LIN {X 0,Y 198.688,Z 628.366,A -85,B 0,C 180,E1 -21497.744,E2 -21497.744} C_VEL
LIN {X 0,Y 197.64,Z 631.779,A -85,B 0,C 180,E1 -21501.82,E2 -21501.82} C_VEL
LIN {X 0,Y 197.241,Z 633.877,A -85,B 0,C 180,E1 -21506.105,E2 -21506.105} C_VEL
LIN {X 0,Y 197.208,Z 634.499,A -85,B 0,C 180,E1 -21509.997,E2 -21509.997} C_VEL
LIN {X 0,Y 197.249,Z 633.864,A -85,B 0,C 180,E1 -21514.084,E2 -21514.084} C_VEL
LIN {X 0,Y 197.637,Z 631.888,A -85,B 0,C 180,E1 -21518.175,E2 -21518.175} C_VEL
LIN {X 0,Y 198.663,Z 628.524,A -85,B 0,C 180,E1 -21522.252,E2 -21522.252} C_VEL
LIN {X 0,Y 200.478,Z 623.671,A -85,B 0,C 180,E1 -21526.284,E2 -21526.284} C_VEL
LIN {X 0,Y 202.386,Z 618.993,A -85,B 0,C 180,E1 -21529.259,E2 -21529.259} C_VEL
LIN {X 0,Y 205.088,Z 612.195,A -85,B 0,C 180,E1 -21532.673,E2 -21532.673} C_VEL
LIN {X 0,Y 208.544,Z 603.751,A -85,B 0,C 180,E1 -21535.98,E2 -21535.98} C_VEL
LIN {X 0,Y 212.007,Z 594.94,A -85,B 0,C 180,E1 -21538.726,E2 -21538.726} C_VEL
LIN {X 0,Y 215.999,Z 584.265,A -85,B 0,C 180,E1 -21541.369,E2 -21541.369} C_VEL
LIN {X 0,Y 219.78,Z 572.903,A -85,B 0,C 180,E1 -21543.607,E2 -21543.607} C_VEL
LIN {X 0,Y 223.02,Z 561.657,A -85,B 0,C 180,E1 -21545.381,E2 -21545.381} C_VEL
LIN {X 0,Y 226.311,Z 548.608,A -85,B 0,C 180,E1 -21546.987,E2 -21546.987} C_VEL
LIN {X 0,Y 228.918,Z 536.079,A -85,B 0,C 180,E1 -21548.157,E2 -21548.157} C_VEL
LIN {X 0,Y 230.973,Z 522.952,A -85,B 0,C 180,E1 -21549.078,E2 -21549.078} C_VEL
LIN {X 0,Y 232.584,Z 508.808,A -85,B 0,C 180,E1 -21549.736,E2 -21549.736} C_VEL
LIN {X 0,Y 236.354,Z 442.048,A -85,B 0,C 180,E1 -21551.632,E2 -21551.632} C_VEL
LIN {X 0,Y 236.321,Z 438.308,A -85,B 0,C 180,E1 -21551.788,E2 -21551.788} C_VEL
LIN {X 0,Y 230.698,Z 425.066,A -85,B 0,C 180,E1 -21553.603,E2 -21553.603} C_VEL
LIN {X 0,Y 225.025,Z 413.286,A -85,B 0,C 180,E1 -21555.516,E2 -21555.516} C_VEL
LIN {X 0,Y 218.681,Z 401.679,A -85,B 0,C 180,E1 -21557.787,E2 -21557.787} C_VEL
LIN {X 0,Y 213.141,Z 392.925,A -85,B 0,C 180,E1 -21559.9,E2 -21559.9} C_VEL
LIN {X 0,Y 210.045,Z 388.672,A -85,B 0,C 180,E1 -21561.139,E2 -21561.139} C_VEL
LIN {X 0,Y 207.427,Z 384.974,A -85,B 0,C 180,E1 -21562.249,E2 -21562.249} C_VEL
LIN {X 0,Y 204.423,Z 381.506,A -85,B 0,C 180,E1 -21563.55,E2 -21563.55} C_VEL
LIN {X 0,Y 203.246,Z 379.556,A -85,B 0,C 180,E1 -21564.116,E2 -21564.116} C_VEL
LIN {X 0,Y 200.84,Z 377.317,A -85,B 0,C 180,E1 -21565.212,E2 -21565.212} C_VEL
LIN {X 0,Y 199.725,Z 374.788,A -85,B 0,C 180,E1 -21566.001,E2 -21566.001} C_VEL
LIN {X 0,Y 199.638,Z 374.276,A -85,B 0,C 180,E1 -21566.514,E2 -21566.514} C_VEL
LIN {X 0,Y 199.656,Z 374.162,A -85,B 0,C 180,E1 -21570.475,E2 -21570.475} C_VEL
LIN {X 0,Y 199.665,Z 374.22,A -85,B 0,C 180,E1 -21575.014,E2 -21575.014} C_VEL
LIN {X 0,Y 199.691,Z 374.213,A -85,B 0,C 180,E1 -21579.394,E2 -21579.394} C_VEL
LIN {X 0,Y 199.795,Z 374.197,A -85,B 0,C 180,E1 -21583.656,E2 -21583.656} C_VEL
LIN {X 0,Y 199.905,Z 374.205,A -85,B 0,C 180,E1 -21587.822,E2 -21587.822} C_VEL
LIN {X 0,Y 200.11,Z 374.161,A -85,B 0,C 180,E1 -21591.924,E2 -21591.924} C_VEL
LIN {X 0,Y 200.314,Z 374.135,A -85,B 0,C 180,E1 -21597.989,E2 -21597.989} C_VEL
LIN {X 0,Y 200.478,Z 374.139,A -85,B 0,C 180,E1 -21600,E2 -21600} C_VEL
LIN {X 0,Y 200.023,Z 374.168,A -85,B 0,C 180,E1 -21604.029,E2 -21604.029} C_VEL
LIN {X 0,Y 200.11,Z 374.161,A -85,B 0,C 180,E1 -21608.076,E2 -21608.076} C_VEL
LIN {X 0,Y 199.904,Z 374.203,A -85,B 0,C 180,E1 -21612.177,E2 -21612.177} C_VEL
LIN {X 0,Y 199.795,Z 374.195,A -85,B 0,C 180,E1 -21616.344,E2 -21616.344} C_VEL
LIN {X 0,Y 199.686,Z 374.214,A -85,B 0,C 180,E1 -21620.001,E2 -21620.001} C_VEL
LIN {X 0,Y 199.025,Z 374.304,A -85,B 0,C 180,E1 -21621.684,E2 -21621.684} C_VEL
LIN {X 0,Y 196.217,Z 374.664,A -85,B 0,C 180,E1 -21624.437,E2 -21624.437} C_VEL
LIN {X 0,Y 192.97,Z 374.996,A -85,B 0,C 180,E1 -21627.849,E2 -21627.849} C_VEL
LIN {X 0,Y 192.61,Z 375.041,A -85,B 0,C 180,E1 -21629.032,E2 -21629.032} C_VEL
LIN {X 0,Y 192.647,Z 375.427,A -85,B 0,C 180,E1 -21630.713,E2 -21630.713} C_VEL
LIN {X 0,Y 193.159,Z 377.057,A -85,B 0,C 180,E1 -21631.383,E2 -21631.383} C_VEL
LIN {X 0,Y 195.117,Z 379.67,A -85,B 0,C 180,E1 -21632.495,E2 -21632.495} C_VEL
LIN {X 0,Y 196.745,Z 380.901,A -85,B 0,C 180,E1 -21633.313,E2 -21633.313} C_VEL
LIN {X 0,Y 198.74,Z 384.113,A -85,B 0,C 180,E1 -21634.381,E2 -21634.381} C_VEL
LIN {X 0,Y 200.861,Z 386.283,A -85,B 0,C 180,E1 -21635.388,E2 -21635.388} C_VEL
LIN {X 0,Y 203.398,Z 389.783,A -85,B 0,C 180,E1 -21636.586,E2 -21636.586} C_VEL
LIN {X 0,Y 204.689,Z 391.4,A -85,B 0,C 180,E1 -21637.163,E2 -21637.163} C_VEL
LIN {X 0,Y 208.318,Z 396.435,A -85,B 0,C 180,E1 -21638.734,E2 -21638.734} C_VEL
LIN {X 0,Y 211.143,Z 400.453,A -85,B 0,C 180,E1 -21639.89,E2 -21639.89} C_VEL
LIN {X 0,Y 217.685,Z 411.697,A -85,B 0,C 180,E1 -21642.451,E2 -21642.451} C_VEL
LIN {X 0,Y 224.176,Z 424.655,A -85,B 0,C 180,E1 -21644.816,E2 -21644.816} C_VEL
LIN {X 0,Y 230.432,Z 439.17,A -85,B 0,C 180,E1 -21646.971,E2 -21646.971} C_VEL
LIN {X 0,Y 231.097,Z 440.853,A -85,B 0,C 180,E1 -21647.195,E2 -21647.195} C_VEL
LIN {X 0,Y 228.019,Z 496.452,A -85,B 0,C 180,E1 -21648.796,E2 -21648.796} C_VEL
LIN {X 0,Y 226.809,Z 513.234,A -85,B 0,C 180,E1 -21649.366,E2 -21649.366} C_VEL
LIN {X 0,Y 224.799,Z 527.804,A -85,B 0,C 180,E1 -21650.144,E2 -21650.144} C_VEL
LIN {X 0,Y 222.26,Z 541.368,A -85,B 0,C 180,E1 -21651.212,E2 -21651.212} C_VEL
LIN {X 0,Y 219.441,Z 553.628,A -85,B 0,C 180,E1 -21652.522,E2 -21652.522} C_VEL
LIN {X 0,Y 216.105,Z 565.698,A -85,B 0,C 180,E1 -21654.173,E2 -21654.173} C_VEL
LIN {X 0,Y 212.305,Z 577.878,A -85,B 0,C 180,E1 -21656.328,E2 -21656.328} C_VEL
LIN {X 0,Y 208.578,Z 587.941,A -85,B 0,C 180,E1 -21658.519,E2 -21658.519} C_VEL
LIN {X 0,Y 204.604,Z 597.944,A -85,B 0,C 180,E1 -21661.26,E2 -21661.26} C_VEL
LIN {X 0,Y 201.059,Z 606.25,A -85,B 0,C 180,E1 -21664.094,E2 -21664.094} C_VEL
LIN {X 0,Y 198.096,Z 613.182,A -85,B 0,C 180,E1 -21667.033,E2 -21667.033} C_VEL
LIN {X 0,Y 195.695,Z 618.917,A -85,B 0,C 180,E1 -21670.055,E2 -21670.055} C_VEL
LIN {X 0,Y 193.677,Z 623.61,A -85,B 0,C 180,E1 -21673.127,E2 -21673.127} C_VEL
LIN {X 0,Y 191.707,Z 628.478,A -85,B 0,C 180,E1 -21677.296,E2 -21677.296} C_VEL
LIN {X 0,Y 190.577,Z 631.857,A -85,B 0,C 180,E1 -21681.52,E2 -21681.52} C_VEL
LIN {X 0,Y 190.163,Z 633.848,A -85,B 0,C 180,E1 -21685.764,E2 -21685.764} C_VEL
LIN {X 0,Y 190.118,Z 634.5,A -85,B 0,C 180,E1 -21690.003,E2 -21690.003} C_VEL
LIN {X 0,Y 190.164,Z 633.824,A -85,B 0,C 180,E1 -21694.242,E2 -21694.242} C_VEL
LIN {X 0,Y 190.734,Z 631.811,A -85,B 0,C 180,E1 -21698.478,E2 -21698.478} C_VEL
LIN {X 0,Y 191.198,Z 630.901,A -85,B 0,C 180,E1 -21700.058,E2 -21700.058} C_VEL
LIN {X 0,Y 192.096,Z 632.211,A -85,B 0,C 180,E1 -21702.683,E2 -21702.683} C_VEL
LIN {X 0,Y 194.442,Z 633.199,A -85,B 0,C 180,E1 -21706.81,E2 -21706.81} C_VEL
LIN {X 0,Y 197.98,Z 632.816,A -85,B 0,C 180,E1 -21710.795,E2 -21710.795} C_VEL
LIN {X 0,Y 202.531,Z 631.063,A -85,B 0,C 180,E1 -21714.611,E2 -21714.611} C_VEL
LIN {X 0,Y 208.298,Z 627.892,A -85,B 0,C 180,E1 -21718.19,E2 -21718.19} C_VEL
LIN {X 0,Y 215.076,Z 623.289,A -85,B 0,C 180,E1 -21721.525,E2 -21721.525} C_VEL
LIN {X 0,Y 222.681,Z 617.112,A -85,B 0,C 180,E1 -21724.62,E2 -21724.62} C_VEL
LIN {X 0,Y 230.147,Z 610.231,A -85,B 0,C 180,E1 -21727.095,E2 -21727.095} C_VEL
LIN {X 0,Y 238.456,Z 601.514,A -85,B 0,C 180,E1 -21729.46,E2 -21729.46} C_VEL
LIN {X 0,Y 246.697,Z 591.63,A -85,B 0,C 180,E1 -21731.482,E2 -21731.482} C_VEL
LIN {X 0,Y 253.123,Z 582.904,A -85,B 0,C 180,E1 -21732.865,E2 -21732.865} C_VEL
LIN {X 0,Y 260.597,Z 571.402,A -85,B 0,C 180,E1 -21734.255,E2 -21734.255} C_VEL
LIN {X 0,Y 267.543,Z 558.852,A -85,B 0,C 180,E1 -21735.409,E2 -21735.409} C_VEL
LIN {X 0,Y 268.161,Z 557.592,A -85,B 0,C 180,E1 -21735.507,E2 -21735.507} C_VEL
LIN {X 0,Y 267.786,Z 558.493,A -85,B 0,C 180,E1 -21735.934,E2 -21735.934} C_VEL
LIN {X 0,Y 261.439,Z 570.62,A -85,B 0,C 180,E1 -21736.936,E2 -21736.936} C_VEL
LIN {X 0,Y 254.824,Z 581.361,A -85,B 0,C 180,E1 -21738.132,E2 -21738.132} C_VEL
LIN {X 0,Y 248.472,Z 590.482,A -85,B 0,C 180,E1 -21739.417,E2 -21739.417} C_VEL
LIN {X 0,Y 240.901,Z 599.981,A -85,B 0,C 180,E1 -21741.154,E2 -21741.154} C_VEL
LIN {X 0,Y 232.636,Z 609.079,A -85,B 0,C 180,E1 -21743.37,E2 -21743.37} C_VEL
LIN {X 0,Y 227.128,Z 614.466,A -85,B 0,C 180,E1 -21745.079,E2 -21745.079} C_VEL
LIN {X 0,Y 220.859,Z 619.969,A -85,B 0,C 180,E1 -21747.251,E2 -21747.251} C_VEL
LIN {X 0,Y 213.286,Z 625.729,A -85,B 0,C 180,E1 -21750.379,E2 -21750.379} C_VEL
LIN {X 0,Y 206.666,Z 629.831,A -85,B 0,C 180,E1 -21753.763,E2 -21753.763} C_VEL
LIN {X 0,Y 203.739,Z 631.338,A -85,B 0,C 180,E1 -21755.547,E2 -21755.547} C_VEL
LIN {X 0,Y 198.992,Z 633.231,A -85,B 0,C 180,E1 -21759.318,E2 -21759.318} C_VEL
LIN {X 0,Y 195.229,Z 633.698,A -85,B 0,C 180,E1 -21763.263,E2 -21763.263} C_VEL
LIN {X 0,Y 192.575,Z 632.768,A -85,B 0,C 180,E1 -21767.352,E2 -21767.352} C_VEL
LIN {X 0,Y 191.078,Z 630.391,A -85,B 0,C 180,E1 -21771.54,E2 -21771.54} C_VEL
LIN {X 0,Y 190.649,Z 626.452,A -85,B 0,C 180,E1 -21775.772,E2 -21775.772} C_VEL
LIN {X 0,Y 190.738,Z 622.348,A -85,B 0,C 180,E1 -21778.945,E2 -21778.945} C_VEL
LIN {X 0,Y 190.954,Z 617.045,A -85,B 0,C 180,E1 -21782.109,E2 -21782.109} C_VEL
LIN {X 0,Y 191.191,Z 610.328,A -85,B 0,C 180,E1 -21785.273,E2 -21785.273} C_VEL
LIN {X 0,Y 191.602,Z 601.884,A -85,B 0,C 180,E1 -21788.437,E2 -21788.437} C_VEL
LIN {X 0,Y 192.123,Z 593.245,A -85,B 0,C 180,E1 -21791.073,E2 -21791.073} C_VEL
LIN {X 0,Y 192.927,Z 582.773,A -85,B 0,C 180,E1 -21793.697,E2 -21793.697} C_VEL
LIN {X 0,Y 193.92,Z 571.144,A -85,B 0,C 180,E1 -21796.042,E2 -21796.042} C_VEL
LIN {X 0,Y 194.965,Z 558.197,A -85,B 0,C 180,E1 -21798.114,E2 -21798.114} C_VEL
LIN {X 0,Y 195.925,Z 544.563,A -85,B 0,C 180,E1 -21799.788,E2 -21799.788} C_VEL
LIN {X 0,Y 196.902,Z 529.324,A -85,B 0,C 180,E1 -21801.134,E2 -21801.134} C_VEL
LIN {X 0,Y 200.175,Z 458.461,A -85,B 0,C 180,E1 -21805.683,E2 -21805.683} C_VEL
LIN {X 0,Y 197.937,Z 429.916,A -85,B 0,C 180,E1 -21807.561,E2 -21807.561} C_VEL
LIN {X 0,Y 197.856,Z 419.514,A -85,B 0,C 180,E1 -21808.293,E2 -21808.293} C_VEL
LIN {X 0,Y 199.54,Z 406.784,A -85,B 0,C 180,E1 -21811.595,E2 -21811.595} C_VEL
LIN {X 0,Y 197.743,Z 398.022,A -85,B 0,C 180,E1 -21814.148,E2 -21814.148} C_VEL
LIN {X 0,Y 197.668,Z 397.343,A -85,B 0,C 180,E1 -21814.672,E2 -21814.672} C_VEL
LIN {X 0,Y 198.255,Z 397.732,A -85,B 0,C 180,E1 -21815.174,E2 -21815.174} C_VEL
LIN {X 0,Y 199.201,Z 398.055,A -85,B 0,C 180,E1 -21815.601,E2 -21815.601} C_VEL
LIN {X 0,Y 201.049,Z 397.617,A -85,B 0,C 180,E1 -21816.305,E2 -21816.305} C_VEL
LIN {X 0,Y 202.414,Z 396.833,A -85,B 0,C 180,E1 -21816.783,E2 -21816.783} C_VEL
LIN {X 0,Y 203.399,Z 397.137,A -85,B 0,C 180,E1 -21817.17,E2 -21817.17} C_VEL
LIN {X 0,Y 206.725,Z 396.78,A -85,B 0,C 180,E1 -21818.351,E2 -21818.351} C_VEL
LIN {X 0,Y 208.167,Z 396.459,A -85,B 0,C 180,E1 -21818.833,E2 -21818.833} C_VEL
LIN {X 0,Y 211.293,Z 400.891,A -85,B 0,C 180,E1 -21820.105,E2 -21820.105} C_VEL
LIN {X 0,Y 217.272,Z 411.228,A -85,B 0,C 180,E1 -21822.442,E2 -21822.442} C_VEL
LIN {X 0,Y 222.993,Z 422.302,A -85,B 0,C 180,E1 -21824.527,E2 -21824.527} C_VEL
LIN {X 0,Y 229.105,Z 435.988,A -85,B 0,C 180,E1 -21826.643,E2 -21826.643} C_VEL
LIN {X 0,Y 230.998,Z 440.808,A -85,B 0,C 180,E1 -21827.285,E2 -21827.285} C_VEL
LIN {X 0,Y 227.011,Z 509.642,A -85,B 0,C 180,E1 -21829.293,E2 -21829.293} C_VEL
LIN {X 0,Y 225.229,Z 524.29,A -85,B 0,C 180,E1 -21830.011,E2 -21830.011} C_VEL
LIN {X 0,Y 222.752,Z 538.201,A -85,B 0,C 180,E1 -21831.018,E2 -21831.018} C_VEL
LIN {X 0,Y 219.914,Z 551.142,A -85,B 0,C 180,E1 -21832.321,E2 -21832.321} C_VEL
LIN {X 0,Y 216.535,Z 563.696,A -85,B 0,C 180,E1 -21833.963,E2 -21833.963} C_VEL
LIN {X 0,Y 212.694,Z 576.322,A -85,B 0,C 180,E1 -21836.108,E2 -21836.108} C_VEL
LIN {X 0,Y 208.627,Z 587.578,A -85,B 0,C 180,E1 -21838.521,E2 -21838.521} C_VEL
LIN {X 0,Y 204.647,Z 597.642,A -85,B 0,C 180,E1 -21841.261,E2 -21841.261} C_VEL
LIN {X 0,Y 201.12,Z 605.999,A -85,B 0,C 180,E1 -21844.097,E2 -21844.097} C_VEL
LIN {X 0,Y 198.086,Z 612.973,A -85,B 0,C 180,E1 -21847.026,E2 -21847.026} C_VEL
LIN {X 0,Y 195.695,Z 618.734,A -85,B 0,C 180,E1 -21850.049,E2 -21850.049} C_VEL
LIN {X 0,Y 193.689,Z 623.467,A -85,B 0,C 180,E1 -21853.123,E2 -21853.123} C_VEL
LIN {X 0,Y 191.72,Z 628.367,A -85,B 0,C 180,E1 -21857.292,E2 -21857.292} C_VEL
LIN {X 0,Y 190.581,Z 631.779,A -85,B 0,C 180,E1 -21861.515,E2 -21861.515} C_VEL
LIN {X 0,Y 190.165,Z 633.807,A -85,B 0,C 180,E1 -21865.758,E2 -21865.758} C_VEL
LIN {X 0,Y 190.119,Z 634.499,A -85,B 0,C 180,E1 -21869.997,E2 -21869.997} C_VEL
LIN {X 0,Y 190.164,Z 633.863,A -85,B 0,C 180,E1 -21874.236,E2 -21874.236} C_VEL
LIN {X 0,Y 190.578,Z 631.888,A -85,B 0,C 180,E1 -21878.48,E2 -21878.48} C_VEL
LIN {X 0,Y 191.697,Z 628.523,A -85,B 0,C 180,E1 -21882.705,E2 -21882.705} C_VEL
LIN {X 0,Y 193.643,Z 623.669,A -85,B 0,C 180,E1 -21886.876,E2 -21886.876} C_VEL
LIN {X 0,Y 196.435,Z 617.183,A -85,B 0,C 180,E1 -21890.961,E2 -21890.961} C_VEL
LIN {X 0,Y 199.479,Z 609.962,A -85,B 0,C 180,E1 -21894.452,E2 -21894.452} C_VEL
LIN {X 0,Y 203.313,Z 601.028,A -85,B 0,C 180,E1 -21897.815,E2 -21897.815} C_VEL
LIN {X 0,Y 207.088,Z 591.645,A -85,B 0,C 180,E1 -21900.598,E2 -21900.598} C_VEL
LIN {X 0,Y 211.056,Z 581.254,A -85,B 0,C 180,E1 -21903.04,E2 -21903.04} C_VEL
LIN {X 0,Y 214.822,Z 569.884,A -85,B 0,C 180,E1 -21905.189,E2 -21905.189} C_VEL
LIN {X 0,Y 218.525,Z 557.084,A -85,B 0,C 180,E1 -21907.083,E2 -21907.083} C_VEL
LIN {X 0,Y 221.531,Z 544.705,A -85,B 0,C 180,E1 -21908.503,E2 -21908.503} C_VEL
LIN {X 0,Y 223.986,Z 532.273,A -85,B 0,C 180,E1 -21909.591,E2 -21909.591} C_VEL
LIN {X 0,Y 226.11,Z 518.478,A -85,B 0,C 180,E1 -21910.451,E2 -21910.451} C_VEL
LIN {X 0,Y 227.577,Z 504,A -85,B 0,C 180,E1 -21911.025,E2 -21911.025} C_VEL
LIN {X 0,Y 231.081,Z 440.795,A -85,B 0,C 180,E1 -21912.856,E2 -21912.856} C_VEL
LIN {X 0,Y 225.276,Z 427.11,A -85,B 0,C 180,E1 -21914.84,E2 -21914.84} C_VEL
LIN {X 0,Y 219.25,Z 414.668,A -85,B 0,C 180,E1 -21917.009,E2 -21917.009} C_VEL
LIN {X 0,Y 212.764,Z 403.025,A -85,B 0,C 180,E1 -21919.504,E2 -21919.504} C_VEL
LIN {X 0,Y 209.554,Z 398.139,A -85,B 0,C 180,E1 -21920.801,E2 -21920.801} C_VEL
LIN {X 0,Y 206.285,Z 393.654,A -85,B 0,C 180,E1 -21922.175,E2 -21922.175} C_VEL
LIN {X 0,Y 203.588,Z 389.967,A -85,B 0,C 180,E1 -21923.376,E2 -21923.376} C_VEL
LIN {X 0,Y 200.923,Z 386.44,A -85,B 0,C 180,E1 -21924.623,E2 -21924.623} C_VEL
LIN {X 0,Y 200.029,Z 385.368,A -85,B 0,C 180,E1 -21925.05,E2 -21925.05} C_VEL
LIN {X 0,Y 197.51,Z 382.418,A -85,B 0,C 180,E1 -21926.298,E2 -21926.298} C_VEL
LIN {X 0,Y 196.601,Z 380.655,A -85,B 0,C 180,E1 -21926.812,E2 -21926.812} C_VEL
LIN {X 0,Y 194.197,Z 378.704,A -85,B 0,C 180,E1 -21928.045,E2 -21928.045} C_VEL
LIN {X 0,Y 192.706,Z 375.703,A -85,B 0,C 180,E1 -21929.145,E2 -21929.145} C_VEL
LIN {X 0,Y 192.613,Z 375.156,A -85,B 0,C 180,E1 -21929.791,E2 -21929.791} C_VEL
LIN {X 0,Y 192.652,Z 375.033,A -85,B 0,C 180,E1 -21931.69,E2 -21931.69} C_VEL
LIN {X 0,Y 192.698,Z 375.105,A -85,B 0,C 180,E1 -21936.347,E2 -21936.347} C_VEL
LIN {X 0,Y 192.723,Z 375.103,A -85,B 0,C 180,E1 -21941.456,E2 -21941.456} C_VEL
LIN {X 0,Y 192.763,Z 375.072,A -85,B 0,C 180,E1 -21945.213,E2 -21945.213} C_VEL
LIN {X 0,Y 192.972,Z 375.045,A -85,B 0,C 180,E1 -21949.508,E2 -21949.508} C_VEL
LIN {X 0,Y 193.059,Z 375.036,A -85,B 0,C 180,E1 -21951.627,E2 -21951.627} C_VEL
LIN {X 0,Y 193.255,Z 375.013,A -85,B 0,C 180,E1 -21957.916,E2 -21957.916} C_VEL
LIN {X 0,Y 193.441,Z 375.015,A -85,B 0,C 180,E1 -21960,E2 -21960} C_VEL
LIN {X 0,Y 192.97,Z 375.046,A -85,B 0,C 180,E1 -21964.177,E2 -21964.177} C_VEL
LIN {X 0,Y 193.059,Z 375.036,A -85,B 0,C 180,E1 -21968.373,E2 -21968.373} C_VEL
LIN {X 0,Y 192.843,Z 375.085,A -85,B 0,C 180,E1 -21972.63,E2 -21972.63} C_VEL
LIN {X 0,Y 192.748,Z 375.077,A -85,B 0,C 180,E1 -21976.959,E2 -21976.959} C_VEL
LIN {X 0,Y 192.627,Z 375.09,A -85,B 0,C 180,E1 -21981.398,E2 -21981.398} C_VEL
LIN {X 0,Y 192.655,Z 375.111,A -85,B 0,C 180,E1 -21984.226,E2 -21984.226} C_VEL
LIN {X 0,Y 192.61,Z 375.041,A -85,B 0,C 180,E1 -21989.032,E2 -21989.032} C_VEL
LIN {X 0,Y 192.786,Z 375.864,A -85,B 0,C 180,E1 -21990.121,E2 -21990.121} C_VEL
LIN {X 0,Y 193.311,Z 377.792,A -85,B 0,C 180,E1 -21991.086,E2 -21991.086} C_VEL
LIN {X 0,Y 194.495,Z 381.894,A -85,B 0,C 180,E1 -21992.313,E2 -21992.313} C_VEL
LIN {X 0,Y 197.836,Z 391.599,A -85,B 0,C 180,E1 -21994.466,E2 -21994.466} C_VEL
LIN {X 0,Y 199.372,Z 394.328,A -85,B 0,C 180,E1 -21995.274,E2 -21995.274} C_VEL
LIN {X 0,Y 200.291,Z 395.434,A -85,B 0,C 180,E1 -21995.712,E2 -21995.712} C_VEL
LIN {X 0,Y 202.195,Z 398.006,A -85,B 0,C 180,E1 -21996.607,E2 -21996.607} C_VEL
LIN {X 0,Y 207.223,Z 405.004,A -85,B 0,C 180,E1 -21998.822,E2 -21998.822} C_VEL
LIN {X 0,Y 213.857,Z 416.694,A -85,B 0,C 180,E1 -22001.565,E2 -22001.565} C_VEL
LIN {X 0,Y 220.02,Z 429.258,A -85,B 0,C 180,E1 -22003.928,E2 -22003.928} C_VEL
LIN {X 0,Y 225.807,Z 443.04,A -85,B 0,C 180,E1 -22006.033,E2 -22006.033} C_VEL
LIN {X 0,Y 222.687,Z 497.061,A -85,B 0,C 180,E1 -22007.609,E2 -22007.609} C_VEL
LIN {X 0,Y 221.385,Z 513.896,A -85,B 0,C 180,E1 -22008.194,E2 -22008.194} C_VEL
LIN {X 0,Y 219.401,Z 527.813,A -85,B 0,C 180,E1 -22008.957,E2 -22008.957} C_VEL
LIN {X 0,Y 216.774,Z 541.375,A -85,B 0,C 180,E1 -22010.037,E2 -22010.037} C_VEL
LIN {X 0,Y 213.848,Z 553.633,A -85,B 0,C 180,E1 -22011.364,E2 -22011.364} C_VEL
LIN {X 0,Y 210.381,Z 565.703,A -85,B 0,C 180,E1 -22013.04,E2 -22013.04} C_VEL
LIN {X 0,Y 206.425,Z 577.881,A -85,B 0,C 180,E1 -22015.234,E2 -22015.234} C_VEL
LIN {X 0,Y 202.552,Z 587.944,A -85,B 0,C 180,E1 -22017.469,E2 -22017.469} C_VEL
LIN {X 0,Y 198.392,Z 597.946,A -85,B 0,C 180,E1 -22020.271,E2 -22020.271} C_VEL
LIN {X 0,Y 194.673,Z 606.251,A -85,B 0,C 180,E1 -22023.178,E2 -22023.178} C_VEL
LIN {X 0,Y 191.541,Z 613.183,A -85,B 0,C 180,E1 -22026.199,E2 -22026.199} C_VEL
LIN {X 0,Y 188.998,Z 618.918,A -85,B 0,C 180,E1 -22029.316,E2 -22029.316} C_VEL
LIN {X 0,Y 186.853,Z 623.612,A -85,B 0,C 180,E1 -22032.491,E2 -22032.491} C_VEL
LIN {X 0,Y 184.761,Z 628.479,A -85,B 0,C 180,E1 -22036.81,E2 -22036.81} C_VEL
LIN {X 0,Y 183.54,Z 631.858,A -85,B 0,C 180,E1 -22041.192,E2 -22041.192} C_VEL
LIN {X 0,Y 183.077,Z 633.848,A -85,B 0,C 180,E1 -22045.6,E2 -22045.6} C_VEL
LIN {X 0,Y 183.031,Z 634.5,A -85,B 0,C 180,E1 -22050.003,E2 -22050.003} C_VEL
LIN {X 0,Y 183.081,Z 633.823,A -85,B 0,C 180,E1 -22054.406,E2 -22054.406} C_VEL
LIN {X 0,Y 183.706,Z 631.811,A -85,B 0,C 180,E1 -22058.805,E2 -22058.805} C_VEL
LIN {X 0,Y 184.385,Z 630.52,A -85,B 0,C 180,E1 -22060.989,E2 -22060.989} C_VEL
LIN {X 0,Y 186.296,Z 632.566,A -85,B 0,C 180,E1 -22065.315,E2 -22065.315} C_VEL
LIN {X 0,Y 189.373,Z 633.278,A -85,B 0,C 180,E1 -22069.515,E2 -22069.515} C_VEL
LIN {X 0,Y 193.629,Z 632.604,A -85,B 0,C 180,E1 -22073.534,E2 -22073.534} C_VEL
LIN {X 0,Y 199.021,Z 630.607,A -85,B 0,C 180,E1 -22077.33,E2 -22077.33} C_VEL
LIN {X 0,Y 205.575,Z 627.261,A -85,B 0,C 180,E1 -22080.853,E2 -22080.853} C_VEL
LIN {X 0,Y 213.093,Z 622.455,A -85,B 0,C 180,E1 -22084.105,E2 -22084.105} C_VEL
LIN {X 0,Y 219.298,Z 617.855,A -85,B 0,C 180,E1 -22086.364,E2 -22086.364} C_VEL
LIN {X 0,Y 228.338,Z 610.157,A -85,B 0,C 180,E1 -22089.124,E2 -22089.124} C_VEL
LIN {X 0,Y 236.859,Z 601.847,A -85,B 0,C 180,E1 -22091.317,E2 -22091.317} C_VEL
LIN {X 0,Y 245.917,Z 591.692,A -85,B 0,C 180,E1 -22093.308,E2 -22093.308} C_VEL
LIN {X 0,Y 252.704,Z 583.019,A -85,B 0,C 180,E1 -22094.609,E2 -22094.609} C_VEL
LIN {X 0,Y 257.75,Z 575.888,A -85,B 0,C 180,E1 -22095.464,E2 -22095.464} C_VEL
LIN {X 0,Y 257.55,Z 576.266,A -85,B 0,C 180,E1 -22095.854,E2 -22095.854} C_VEL
LIN {X 0,Y 250.06,Z 587.04,A -85,B 0,C 180,E1 -22097.146,E2 -22097.146} C_VEL
LIN {X 0,Y 240.926,Z 598.26,A -85,B 0,C 180,E1 -22098.978,E2 -22098.978} C_VEL
LIN {X 0,Y 233.307,Z 606.377,A -85,B 0,C 180,E1 -22100.758,E2 -22100.758} C_VEL
LIN {X 0,Y 226.064,Z 613.211,A -85,B 0,C 180,E1 -22102.683,E2 -22102.683} C_VEL
LIN {X 0,Y 217.205,Z 620.508,A -85,B 0,C 180,E1 -22105.512,E2 -22105.512} C_VEL
LIN {X 0,Y 209.15,Z 626.051,A -85,B 0,C 180,E1 -22108.611,E2 -22108.611} C_VEL
LIN {X 0,Y 203.76,Z 629.173,A -85,B 0,C 180,E1 -22111.126,E2 -22111.126} C_VEL
LIN {X 0,Y 197.33,Z 632.035,A -85,B 0,C 180,E1 -22114.698,E2 -22114.698} C_VEL
LIN {X 0,Y 192.364,Z 633.49,A -85,B 0,C 180,E1 -22118.571,E2 -22118.571} C_VEL
LIN {X 0,Y 188.455,Z 633.576,A -85,B 0,C 180,E1 -22122.642,E2 -22122.642} C_VEL
LIN {X 0,Y 185.681,Z 632.233,A -85,B 0,C 180,E1 -22126.874,E2 -22126.874} C_VEL
LIN {X 0,Y 184.109,Z 629.491,A -85,B 0,C 180,E1 -22131.217,E2 -22131.217} C_VEL
LIN {X 0,Y 183.687,Z 625.204,A -85,B 0,C 180,E1 -22135.612,E2 -22135.612} C_VEL
LIN {X 0,Y 183.808,Z 620.821,A -85,B 0,C 180,E1 -22138.905,E2 -22138.905} C_VEL
LIN {X 0,Y 184.04,Z 615.199,A -85,B 0,C 180,E1 -22142.189,E2 -22142.189} C_VEL
LIN {X 0,Y 184.297,Z 608.108,A -85,B 0,C 180,E1 -22145.451,E2 -22145.451} C_VEL
LIN {X 0,Y 184.65,Z 600.307,A -85,B 0,C 180,E1 -22148.368,E2 -22148.368} C_VEL
LIN {X 0,Y 185.151,Z 591.98,A -85,B 0,C 180,E1 -22150.941,E2 -22150.941} C_VEL
LIN {X 0,Y 185.975,Z 581.266,A -85,B 0,C 180,E1 -22153.662,E2 -22153.662} C_VEL
LIN {X 0,Y 186.981,Z 569.447,A -85,B 0,C 180,E1 -22156.093,E2 -22156.093} C_VEL
LIN {X 0,Y 188.035,Z 556.02,A -85,B 0,C 180,E1 -22158.242,E2 -22158.242} C_VEL
LIN {X 0,Y 188.93,Z 543.01,A -85,B 0,C 180,E1 -22159.843,E2 -22159.843} C_VEL
LIN {X 0,Y 189.852,Z 528.449,A -85,B 0,C 180,E1 -22161.157,E2 -22161.157} C_VEL
LIN {X 0,Y 193.065,Z 458.287,A -85,B 0,C 180,E1 -22165.884,E2 -22165.884} C_VEL
LIN {X 0,Y 190.927,Z 431.154,A -85,B 0,C 180,E1 -22167.752,E2 -22167.752} C_VEL
LIN {X 0,Y 190.801,Z 419.734,A -85,B 0,C 180,E1 -22168.549,E2 -22168.549} C_VEL
LIN {X 0,Y 192.452,Z 407.164,A -85,B 0,C 180,E1 -22171.929,E2 -22171.929} C_VEL
LIN {X 0,Y 192.198,Z 405.757,A -85,B 0,C 180,E1 -22172.505,E2 -22172.505} C_VEL
LIN {X 0,Y 192.386,Z 405.607,A -85,B 0,C 180,E1 -22173.096,E2 -22173.096} C_VEL
LIN {X 0,Y 193.318,Z 406.18,A -85,B 0,C 180,E1 -22173.624,E2 -22173.624} C_VEL
LIN {X 0,Y 195.047,Z 405.896,A -85,B 0,C 180,E1 -22174.363,E2 -22174.363} C_VEL
LIN {X 0,Y 196.485,Z 404.925,A -85,B 0,C 180,E1 -22174.911,E2 -22174.911} C_VEL
LIN {X 0,Y 201.135,Z 404.586,A -85,B 0,C 180,E1 -22176.748,E2 -22176.748} C_VEL
LIN {X 0,Y 206.038,Z 403.924,A -85,B 0,C 180,E1 -22178.502,E2 -22178.502} C_VEL
LIN {X 0,Y 206.908,Z 404.71,A -85,B 0,C 180,E1 -22178.847,E2 -22178.847} C_VEL
LIN {X 0,Y 213.149,Z 415.575,A -85,B 0,C 180,E1 -22181.432,E2 -22181.432} C_VEL
LIN {X 0,Y 219.179,Z 427.617,A -85,B 0,C 180,E1 -22183.751,E2 -22183.751} C_VEL
LIN {X 0,Y 224.789,Z 440.662,A -85,B 0,C 180,E1 -22185.799,E2 -22185.799} C_VEL
LIN {X 0,Y 225.704,Z 442.949,A -85,B 0,C 180,E1 -22186.123,E2 -22186.123} C_VEL
LIN {X 0,Y 221.672,Z 509.843,A -85,B 0,C 180,E1 -22188.107,E2 -22188.107} C_VEL
LIN {X 0,Y 219.846,Z 524.3,A -85,B 0,C 180,E1 -22188.824,E2 -22188.824} C_VEL
LIN {X 0,Y 217.283,Z 538.209,A -85,B 0,C 180,E1 -22189.841,E2 -22189.841} C_VEL
LIN {X 0,Y 214.346,Z 551.147,A -85,B 0,C 180,E1 -22191.163,E2 -22191.163} C_VEL
LIN {X 0,Y 210.824,Z 563.701,A -85,B 0,C 180,E1 -22192.825,E2 -22192.825} C_VEL
LIN {X 0,Y 207.209,Z 575.152,A -85,B 0,C 180,E1 -22194.786,E2 -22194.786} C_VEL
LIN {X 0,Y 203.369,Z 585.663,A -85,B 0,C 180,E1 -22197.022,E2 -22197.022} C_VEL
LIN {X 0,Y 199.076,Z 596.105,A -85,B 0,C 180,E1 -22199.794,E2 -22199.794} C_VEL
LIN {X 0,Y 195.323,Z 604.719,A -85,B 0,C 180,E1 -22202.69,E2 -22202.69} C_VEL
LIN {X 0,Y 191.545,Z 612.975,A -85,B 0,C 180,E1 -22206.194,E2 -22206.194} C_VEL
LIN {X 0,Y 188.988,Z 618.735,A -85,B 0,C 180,E1 -22209.309,E2 -22209.309} C_VEL
LIN {X 0,Y 186.865,Z 623.468,A -85,B 0,C 180,E1 -22212.487,E2 -22212.487} C_VEL
LIN {X 0,Y 184.775,Z 628.368,A -85,B 0,C 180,E1 -22216.805,E2 -22216.805} C_VEL
LIN {X 0,Y 183.545,Z 631.78,A -85,B 0,C 180,E1 -22221.187,E2 -22221.187} C_VEL
LIN {X 0,Y 183.08,Z 633.807,A -85,B 0,C 180,E1 -22225.594,E2 -22225.594} C_VEL
LIN {X 0,Y 183.032,Z 634.499,A -85,B 0,C 180,E1 -22229.997,E2 -22229.997} C_VEL
LIN {X 0,Y 183.078,Z 633.863,A -85,B 0,C 180,E1 -22234.4,E2 -22234.4} C_VEL
LIN {X 0,Y 183.541,Z 631.887,A -85,B 0,C 180,E1 -22238.807,E2 -22238.807} C_VEL
LIN {X 0,Y 184.753,Z 628.522,A -85,B 0,C 180,E1 -22243.19,E2 -22243.19} C_VEL
LIN {X 0,Y 186.822,Z 623.668,A -85,B 0,C 180,E1 -22247.512,E2 -22247.512} C_VEL
LIN {X 0,Y 189.778,Z 617.181,A -85,B 0,C 180,E1 -22251.733,E2 -22251.733} C_VEL
LIN {X 0,Y 192.999,Z 609.96,A -85,B 0,C 180,E1 -22255.329,E2 -22255.329} C_VEL
LIN {X 0,Y 197.026,Z 601.026,A -85,B 0,C 180,E1 -22258.784,E2 -22258.784} C_VEL
LIN {X 0,Y 200.996,Z 591.642,A -85,B 0,C 180,E1 -22261.63,E2 -22261.63} C_VEL
LIN {X 0,Y 205.137,Z 581.25,A -85,B 0,C 180,E1 -22264.122,E2 -22264.122} C_VEL
LIN {X 0,Y 209.245,Z 569.229,A -85,B 0,C 180,E1 -22266.423,E2 -22266.423} C_VEL
LIN {X 0,Y 212.906,Z 557.079,A -85,B 0,C 180,E1 -22268.235,E2 -22268.235} C_VEL
LIN {X 0,Y 216.027,Z 544.698,A -85,B 0,C 180,E1 -22269.674,E2 -22269.674} C_VEL
LIN {X 0,Y 218.565,Z 532.264,A -85,B 0,C 180,E1 -22270.776,E2 -22270.776} C_VEL
LIN {X 0,Y 220.762,Z 518.466,A -85,B 0,C 180,E1 -22271.645,E2 -22271.645} C_VEL
LIN {X 0,Y 222.204,Z 504.869,A -85,B 0,C 180,E1 -22272.197,E2 -22272.197} C_VEL
LIN {X 0,Y 225.792,Z 442.971,A -85,B 0,C 180,E1 -22274.019,E2 -22274.019} C_VEL
LIN {X 0,Y 219.329,Z 427.753,A -85,B 0,C 180,E1 -22276.375,E2 -22276.375} C_VEL
LIN {X 0,Y 213.023,Z 415.138,A -85,B 0,C 180,E1 -22278.812,E2 -22278.812} C_VEL
LIN {X 0,Y 206.98,Z 404.574,A -85,B 0,C 180,E1 -22281.331,E2 -22281.331} C_VEL
LIN {X 0,Y 200.609,Z 395.795,A -85,B 0,C 180,E1 -22284.185,E2 -22284.185} C_VEL
LIN {X 0,Y 197.075,Z 391.191,A -85,B 0,C 180,E1 -22285.925,E2 -22285.925} C_VEL
LIN {X 0,Y 194.498,Z 387.893,A -85,B 0,C 180,E1 -22287.283,E2 -22287.283} C_VEL
LIN {X 0,Y 193.565,Z 386.609,A -85,B 0,C 180,E1 -22287.802,E2 -22287.802} C_VEL
LIN {X 0,Y 191.222,Z 384.154,A -85,B 0,C 180,E1 -22289.11,E2 -22289.11} C_VEL
LIN {X 0,Y 189.818,Z 381.639,A -85,B 0,C 180,E1 -22290.011,E2 -22290.011} C_VEL
LIN {X 0,Y 187.243,Z 379.638,A -85,B 0,C 180,E1 -22291.561,E2 -22291.561} C_VEL
LIN {X 0,Y 185.659,Z 376.641,A -85,B 0,C 180,E1 -22292.907,E2 -22292.907} C_VEL
LIN {X 0,Y 185.566,Z 376.047,A -85,B 0,C 180,E1 -22293.576,E2 -22293.576} C_VEL
LIN {X 0,Y 185.588,Z 375.972,A -85,B 0,C 180,E1 -22297.747,E2 -22297.747} C_VEL
LIN {X 0,Y 185.681,Z 375.968,A -85,B 0,C 180,E1 -22302.374,E2 -22302.374} C_VEL
LIN {X 0,Y 185.755,Z 375.962,A -85,B 0,C 180,E1 -22306.879,E2 -22306.879} C_VEL
LIN {X 0,Y 186.005,Z 375.912,A -85,B 0,C 180,E1 -22311.307,E2 -22311.307} C_VEL
LIN {X 0,Y 186.2,Z 375.89,A -85,B 0,C 180,E1 -22317.837,E2 -22317.837} C_VEL
LIN {X 0,Y 186.403,Z 375.892,A -85,B 0,C 180,E1 -22320,E2 -22320} C_VEL
LIN {X 0,Y 185.917,Z 375.925,A -85,B 0,C 180,E1 -22324.336,E2 -22324.336} C_VEL
LIN {X 0,Y 186.005,Z 375.911,A -85,B 0,C 180,E1 -22328.693,E2 -22328.693} C_VEL
LIN {X 0,Y 185.755,Z 375.961,A -85,B 0,C 180,E1 -22333.121,E2 -22333.121} C_VEL
LIN {X 0,Y 185.666,Z 375.975,A -85,B 0,C 180,E1 -22338.868,E2 -22338.868} C_VEL
LIN {X 0,Y 185.587,Z 375.97,A -85,B 0,C 180,E1 -22342.252,E2 -22342.252} C_VEL
LIN {X 0,Y 185.564,Z 376.112,A -85,B 0,C 180,E1 -22346.575,E2 -22346.575} C_VEL
LIN {X 0,Y 185.75,Z 376.928,A -85,B 0,C 180,E1 -22347.307,E2 -22347.307} C_VEL
LIN {X 0,Y 187.373,Z 379.805,A -85,B 0,C 180,E1 -22348.57,E2 -22348.57} C_VEL
LIN {X 0,Y 190.044,Z 382.011,A -85,B 0,C 180,E1 -22350.179,E2 -22350.179} C_VEL
LIN {X 0,Y 192.092,Z 385.297,A -85,B 0,C 180,E1 -22351.446,E2 -22351.446} C_VEL
LIN {X 0,Y 194.234,Z 387.421,A -85,B 0,C 180,E1 -22352.609,E2 -22352.609} C_VEL
LIN {X 0,Y 196.814,Z 390.937,A -85,B 0,C 180,E1 -22353.991,E2 -22353.991} C_VEL
LIN {X 0,Y 198.246,Z 392.661,A -85,B 0,C 180,E1 -22354.709,E2 -22354.709} C_VEL
LIN {X 0,Y 200.291,Z 395.434,A -85,B 0,C 180,E1 -22355.712,E2 -22355.712} C_VEL
LIN {X 0,Y 201.562,Z 397.5,A -85,B 0,C 180,E1 -22356.334,E2 -22356.334} C_VEL
LIN {X 0,Y 202.651,Z 401.424,A -85,B 0,C 180,E1 -22356.978,E2 -22356.978} C_VEL
LIN {X 0,Y 204.211,Z 410.108,A -85,B 0,C 180,E1 -22358.044,E2 -22358.044} C_VEL
LIN {X 0,Y 205.522,Z 413.208,A -85,B 0,C 180,E1 -22358.68,E2 -22358.68} C_VEL
LIN {X 0,Y 211.753,Z 424.978,A -85,B 0,C 180,E1 -22361.337,E2 -22361.337} C_VEL
LIN {X 0,Y 217.721,Z 438.05,A -85,B 0,C 180,E1 -22363.708,E2 -22363.708} C_VEL
LIN {X 0,Y 220.676,Z 445.441,A -85,B 0,C 180,E1 -22364.841,E2 -22364.841} C_VEL
LIN {X 0,Y 217.39,Z 498.672,A -85,B 0,C 180,E1 -22366.393,E2 -22366.393} C_VEL
LIN {X 0,Y 216.159,Z 513.91,A -85,B 0,C 180,E1 -22366.943,E2 -22366.943} C_VEL
LIN {X 0,Y 214.108,Z 527.822,A -85,B 0,C 180,E1 -22367.712,E2 -22367.712} C_VEL
LIN {X 0,Y 211.387,Z 541.382,A -85,B 0,C 180,E1 -22368.802,E2 -22368.802} C_VEL
LIN {X 0,Y 208.335,Z 553.638,A -85,B 0,C 180,E1 -22370.141,E2 -22370.141} C_VEL
LIN {X 0,Y 204.735,Z 565.707,A -85,B 0,C 180,E1 -22371.841,E2 -22371.841} C_VEL
LIN {X 0,Y 200.619,Z 577.885,A -85,B 0,C 180,E1 -22374.075,E2 -22374.075} C_VEL
LIN {X 0,Y 196.603,Z 587.947,A -85,B 0,C 180,E1 -22376.356,E2 -22376.356} C_VEL
LIN {X 0,Y 192.224,Z 597.949,A -85,B 0,C 180,E1 -22379.216,E2 -22379.216} C_VEL
LIN {X 0,Y 188.344,Z 606.253,A -85,B 0,C 180,E1 -22382.2,E2 -22382.2} C_VEL
LIN {X 0,Y 185.015,Z 613.185,A -85,B 0,C 180,E1 -22385.304,E2 -22385.304} C_VEL
LIN {X 0,Y 182.336,Z 618.919,A -85,B 0,C 180,E1 -22388.524,E2 -22388.524} C_VEL
LIN {X 0,Y 180.061,Z 623.613,A -85,B 0,C 180,E1 -22391.808,E2 -22391.808} C_VEL
LIN {X 0,Y 177.832,Z 628.48,A -85,B 0,C 180,E1 -22396.286,E2 -22396.286} C_VEL
LIN {X 0,Y 176.498,Z 631.858,A -85,B 0,C 180,E1 -22400.838,E2 -22400.838} C_VEL
LIN {X 0,Y 176.007,Z 633.849,A -85,B 0,C 180,E1 -22405.422,E2 -22405.422} C_VEL
LIN {X 0,Y 175.945,Z 634.5,A -85,B 0,C 180,E1 -22410.003,E2 -22410.003} C_VEL
LIN {X 0,Y 176.012,Z 633.823,A -85,B 0,C 180,E1 -22414.583,E2 -22414.583} C_VEL
LIN {X 0,Y 176.679,Z 631.81,A -85,B 0,C 180,E1 -22419.158,E2 -22419.158} C_VEL
LIN {X 0,Y 177.625,Z 630.086,A -85,B 0,C 180,E1 -22421.992,E2 -22421.992} C_VEL
LIN {X 0,Y 179.453,Z 632.136,A -85,B 0,C 180,E1 -22425.914,E2 -22425.914} C_VEL
LIN {X 0,Y 182.68,Z 633.209,A -85,B 0,C 180,E1 -22430.261,E2 -22430.261} C_VEL
LIN {X 0,Y 187.141,Z 632.982,A -85,B 0,C 180,E1 -22434.402,E2 -22434.402} C_VEL
LIN {X 0,Y 192.794,Z 631.466,A -85,B 0,C 180,E1 -22438.29,E2 -22438.29} C_VEL
LIN {X 0,Y 199.633,Z 628.627,A -85,B 0,C 180,E1 -22441.878,E2 -22441.878} C_VEL
LIN {X 0,Y 207.452,Z 624.368,A -85,B 0,C 180,E1 -22445.167,E2 -22445.167} C_VEL
LIN {X 0,Y 213.865,Z 620.237,A -85,B 0,C 180,E1 -22447.444,E2 -22447.444} C_VEL
LIN {X 0,Y 220.848,Z 615.184,A -85,B 0,C 180,E1 -22449.531,E2 -22449.531} C_VEL
LIN {X 0,Y 229.488,Z 608.008,A -85,B 0,C 180,E1 -22451.768,E2 -22451.768} C_VEL
LIN {X 0,Y 238.624,Z 599.345,A -85,B 0,C 180,E1 -22453.801,E2 -22453.801} C_VEL
LIN {X 0,Y 246.87,Z 590.4,A -85,B 0,C 180,E1 -22455.377,E2 -22455.377} C_VEL
LIN {X 0,Y 247.185,Z 590.08,A -85,B 0,C 180,E1 -22455.805,E2 -22455.805} C_VEL
LIN {X 0,Y 238.705,Z 599.65,A -85,B 0,C 180,E1 -22457.377,E2 -22457.377} C_VEL
LIN {X 0,Y 229.461,Z 608.666,A -85,B 0,C 180,E1 -22459.394,E2 -22459.394} C_VEL
LIN {X 0,Y 220.755,Z 615.988,A -85,B 0,C 180,E1 -22461.625,E2 -22461.625} C_VEL
LIN {X 0,Y 211.585,Z 622.578,A -85,B 0,C 180,E1 -22464.46,E2 -22464.46} C_VEL
LIN {X 0,Y 205.26,Z 626.44,A -85,B 0,C 180,E1 -22466.782,E2 -22466.782} C_VEL
LIN {X 0,Y 197.64,Z 630.273,A -85,B 0,C 180,E1 -22470.143,E2 -22470.143} C_VEL
LIN {X 0,Y 190.966,Z 632.644,A -85,B 0,C 180,E1 -22473.792,E2 -22473.792} C_VEL
LIN {X 0,Y 185.767,Z 633.629,A -85,B 0,C 180,E1 -22477.77,E2 -22477.77} C_VEL
LIN {X 0,Y 181.707,Z 633.294,A -85,B 0,C 180,E1 -22481.976,E2 -22481.976} C_VEL
LIN {X 0,Y 178.806,Z 631.599,A -85,B 0,C 180,E1 -22486.36,E2 -22486.36} C_VEL
LIN {X 0,Y 177.182,Z 628.449,A -85,B 0,C 180,E1 -22490.871,E2 -22490.871} C_VEL
LIN {X 0,Y 176.746,Z 625.692,A -85,B 0,C 180,E1 -22493.786,E2 -22493.786} C_VEL
LIN {X 0,Y 176.85,Z 620.809,A -85,B 0,C 180,E1 -22497.723,E2 -22497.723} C_VEL
LIN {X 0,Y 177.065,Z 615.311,A -85,B 0,C 180,E1 -22501.137,E2 -22501.137} C_VEL
LIN {X 0,Y 177.284,Z 609.617,A -85,B 0,C 180,E1 -22503.978,E2 -22503.978} C_VEL
LIN {X 0,Y 177.568,Z 602.741,A -85,B 0,C 180,E1 -22506.819,E2 -22506.819} C_VEL
LIN {X 0,Y 178.064,Z 592.492,A -85,B 0,C 180,E1 -22510.231,E2 -22510.231} C_VEL
LIN {X 0,Y 178.841,Z 582.021,A -85,B 0,C 180,E1 -22513.06,E2 -22513.06} C_VEL
LIN {X 0,Y 179.796,Z 570.393,A -85,B 0,C 180,E1 -22515.589,E2 -22515.589} C_VEL
LIN {X 0,Y 180.676,Z 559.206,A -85,B 0,C 180,E1 -22517.546,E2 -22517.546} C_VEL
LIN {X 0,Y 181.59,Z 546.069,A -85,B 0,C 180,E1 -22519.353,E2 -22519.353} C_VEL
LIN {X 0,Y 182.516,Z 532.038,A -85,B 0,C 180,E1 -22520.792,E2 -22520.792} C_VEL
LIN {X 0,Y 184.144,Z 496.435,A -85,B 0,C 180,E1 -22523.394,E2 -22523.394} C_VEL
LIN {X 0,Y 185.939,Z 458.528,A -85,B 0,C 180,E1 -22526.047,E2 -22526.047} C_VEL
LIN {X 0,Y 183.835,Z 429.462,A -85,B 0,C 180,E1 -22528.136,E2 -22528.136} C_VEL
LIN {X 0,Y 183.839,Z 420.238,A -85,B 0,C 180,E1 -22528.911,E2 -22528.911} C_VEL
LIN {X 0,Y 184.073,Z 418.664,A -85,B 0,C 180,E1 -22529.34,E2 -22529.34} C_VEL
LIN {X 0,Y 184.673,Z 417.647,A -85,B 0,C 180,E1 -22530.124,E2 -22530.124} C_VEL
LIN {X 0,Y 186.336,Z 417.528,A -85,B 0,C 180,E1 -22531.081,E2 -22531.081} C_VEL
LIN {X 0,Y 189.119,Z 415.383,A -85,B 0,C 180,E1 -22532.305,E2 -22532.305} C_VEL
LIN {X 0,Y 191.192,Z 413.115,A -85,B 0,C 180,E1 -22533.123,E2 -22533.123} C_VEL
LIN {X 0,Y 194.668,Z 413.008,A -85,B 0,C 180,E1 -22534.654,E2 -22534.654} C_VEL
LIN {X 0,Y 196.793,Z 411.938,A -85,B 0,C 180,E1 -22535.474,E2 -22535.474} C_VEL
LIN {X 0,Y 201.258,Z 411.509,A -85,B 0,C 180,E1 -22537.197,E2 -22537.197} C_VEL
LIN {X 0,Y 202.084,Z 411.237,A -85,B 0,C 180,E1 -22537.489,E2 -22537.489} C_VEL
LIN {X 0,Y 204.335,Z 411.452,A -85,B 0,C 180,E1 -22538.317,E2 -22538.317} C_VEL
LIN {X 0,Y 209.78,Z 421.363,A -85,B 0,C 180,E1 -22540.676,E2 -22540.676} C_VEL
LIN {X 0,Y 215.411,Z 432.909,A -85,B 0,C 180,E1 -22542.947,E2 -22542.947} C_VEL
LIN {X 0,Y 220.498,Z 445.202,A -85,B 0,C 180,E1 -22544.909,E2 -22544.909} C_VEL
LIN {X 0,Y 216.434,Z 510.043,A -85,B 0,C 180,E1 -22546.864,E2 -22546.864} C_VEL
LIN {X 0,Y 214.562,Z 524.31,A -85,B 0,C 180,E1 -22547.578,E2 -22547.578} C_VEL
LIN {X 0,Y 211.908,Z 538.216,A -85,B 0,C 180,E1 -22548.603,E2 -22548.603} C_VEL
LIN {X 0,Y 208.868,Z 551.153,A -85,B 0,C 180,E1 -22549.943,E2 -22549.943} C_VEL
LIN {X 0,Y 205.196,Z 563.705,A -85,B 0,C 180,E1 -22551.624,E2 -22551.624} C_VEL
LIN {X 0,Y 201.432,Z 575.156,A -85,B 0,C 180,E1 -22553.618,E2 -22553.618} C_VEL
LIN {X 0,Y 197.443,Z 585.666,A -85,B 0,C 180,E1 -22555.898,E2 -22555.898} C_VEL
LIN {X 0,Y 192.947,Z 596.108,A -85,B 0,C 180,E1 -22558.729,E2 -22558.729} C_VEL
LIN {X 0,Y 189.025,Z 604.722,A -85,B 0,C 180,E1 -22561.7,E2 -22561.7} C_VEL
LIN {X 0,Y 185.026,Z 612.977,A -85,B 0,C 180,E1 -22565.3,E2 -22565.3} C_VEL
LIN {X 0,Y 182.321,Z 618.737,A -85,B 0,C 180,E1 -22568.516,E2 -22568.516} C_VEL
LIN {X 0,Y 180.074,Z 623.469,A -85,B 0,C 180,E1 -22571.804,E2 -22571.804} C_VEL
LIN {X 0,Y 177.847,Z 628.369,A -85,B 0,C 180,E1 -22576.282,E2 -22576.282} C_VEL
LIN {X 0,Y 176.502,Z 631.78,A -85,B 0,C 180,E1 -22580.832,E2 -22580.832} C_VEL
LIN {X 0,Y 176.01,Z 633.807,A -85,B 0,C 180,E1 -22585.417,E2 -22585.417} C_VEL
LIN {X 0,Y 175.946,Z 634.499,A -85,B 0,C 180,E1 -22589.997,E2 -22589.997} C_VEL
LIN {X 0,Y 176.008,Z 633.863,A -85,B 0,C 180,E1 -22594.578,E2 -22594.578} C_VEL
LIN {X 0,Y 176.498,Z 631.887,A -85,B 0,C 180,E1 -22599.162,E2 -22599.162} C_VEL
LIN {X 0,Y 177.826,Z 628.521,A -85,B 0,C 180,E1 -22603.714,E2 -22603.714} C_VEL
LIN {X 0,Y 180.032,Z 623.667,A -85,B 0,C 180,E1 -22608.195,E2 -22608.195} C_VEL
LIN {X 0,Y 183.143,Z 617.18,A -85,B 0,C 180,E1 -22612.563,E2 -22612.563} C_VEL
LIN {X 0,Y 186.563,Z 609.959,A -85,B 0,C 180,E1 -22616.269,E2 -22616.269} C_VEL
LIN {X 0,Y 190.8,Z 601.024,A -85,B 0,C 180,E1 -22619.816,E2 -22619.816} C_VEL
LIN {X 0,Y 194.982,Z 591.639,A -85,B 0,C 180,E1 -22622.725,E2 -22622.725} C_VEL
LIN {X 0,Y 199.287,Z 581.247,A -85,B 0,C 180,E1 -22625.27,E2 -22625.27} C_VEL
LIN {X 0,Y 203.341,Z 569.91,A -85,B 0,C 180,E1 -22627.495,E2 -22627.495} C_VEL
LIN {X 0,Y 207.356,Z 557.074,A -85,B 0,C 180,E1 -22629.453,E2 -22629.453} C_VEL
LIN {X 0,Y 210.616,Z 544.692,A -85,B 0,C 180,E1 -22630.906,E2 -22630.906} C_VEL
LIN {X 0,Y 213.481,Z 530.955,A -85,B 0,C 180,E1 -22632.122,E2 -22632.122} C_VEL
LIN {X 0,Y 215.788,Z 516.625,A -85,B 0,C 180,E1 -22632.99,E2 -22632.99} C_VEL
LIN {X 0,Y 217.177,Z 502.707,A -85,B 0,C 180,E1 -22633.525,E2 -22633.525} C_VEL
LIN {X 0,Y 220.62,Z 445.224,A -85,B 0,C 180,E1 -22635.228,E2 -22635.228} C_VEL
LIN {X 0,Y 214.375,Z 430.543,A -85,B 0,C 180,E1 -22637.645,E2 -22637.645} C_VEL
LIN {X 0,Y 208.923,Z 419.473,A -85,B 0,C 180,E1 -22639.885,E2 -22639.885} C_VEL
LIN {X 0,Y 203.484,Z 409.846,A -85,B 0,C 180,E1 -22642.278,E2 -22642.278} C_VEL
LIN {X 0,Y 197.5,Z 401.362,A -85,B 0,C 180,E1 -22645.105,E2 -22645.105} C_VEL
LIN {X 0,Y 194.091,Z 396.887,A -85,B 0,C 180,E1 -22646.87,E2 -22646.87} C_VEL
LIN {X 0,Y 190.999,Z 392.755,A -85,B 0,C 180,E1 -22648.608,E2 -22648.608} C_VEL
LIN {X 0,Y 188.319,Z 389.551,A -85,B 0,C 180,E1 -22650.21,E2 -22650.21} C_VEL
LIN {X 0,Y 187.229,Z 387.898,A -85,B 0,C 180,E1 -22650.925,E2 -22650.925} C_VEL
LIN {X 0,Y 184.554,Z 385.266,A -85,B 0,C 180,E1 -22652.671,E2 -22652.671} C_VEL
LIN {X 0,Y 183.079,Z 382.664,A -85,B 0,C 180,E1 -22653.803,E2 -22653.803} C_VEL
LIN {X 0,Y 180.241,Z 380.683,A -85,B 0,C 180,E1 -22655.887,E2 -22655.887} C_VEL
LIN {X 0,Y 178.857,Z 378.322,A -85,B 0,C 180,E1 -22657.168,E2 -22657.168} C_VEL
LIN {X 0,Y 178.615,Z 377.309,A -85,B 0,C 180,E1 -22657.745,E2 -22657.745} C_VEL
LIN {X 0,Y 178.546,Z 376.9,A -85,B 0,C 180,E1 -22658.647,E2 -22658.647} C_VEL
LIN {X 0,Y 178.641,Z 376.856,A -85,B 0,C 180,E1 -22661.655,E2 -22661.655} C_VEL
LIN {X 0,Y 178.672,Z 376.836,A -85,B 0,C 180,E1 -22666.349,E2 -22666.349} C_VEL
LIN {X 0,Y 178.954,Z 376.788,A -85,B 0,C 180,E1 -22670.962,E2 -22670.962} C_VEL
LIN {X 0,Y 179.145,Z 376.768,A -85,B 0,C 180,E1 -22677.751,E2 -22677.751} C_VEL
LIN {X 0,Y 179.366,Z 376.769,A -85,B 0,C 180,E1 -22680,E2 -22680} C_VEL
LIN {X 0,Y 178.866,Z 376.804,A -85,B 0,C 180,E1 -22684.507,E2 -22684.507} C_VEL
LIN {X 0,Y 178.954,Z 376.787,A -85,B 0,C 180,E1 -22689.038,E2 -22689.038} C_VEL
LIN {X 0,Y 178.672,Z 376.834,A -85,B 0,C 180,E1 -22693.651,E2 -22693.651} C_VEL
LIN {X 0,Y 178.614,Z 376.848,A -85,B 0,C 180,E1 -22699.217,E2 -22699.217} C_VEL
LIN {X 0,Y 178.595,Z 377.183,A -85,B 0,C 180,E1 -22702.105,E2 -22702.105} C_VEL
LIN {X 0,Y 178.88,Z 378.397,A -85,B 0,C 180,E1 -22702.905,E2 -22702.905} C_VEL
LIN {X 0,Y 180.408,Z 380.861,A -85,B 0,C 180,E1 -22704.292,E2 -22704.292} C_VEL
LIN {X 0,Y 183.282,Z 382.951,A -85,B 0,C 180,E1 -22706.395,E2 -22706.395} C_VEL
LIN {X 0,Y 185.209,Z 386.128,A -85,B 0,C 180,E1 -22707.833,E2 -22707.833} C_VEL
LIN {X 0,Y 187.692,Z 388.468,A -85,B 0,C 180,E1 -22709.417,E2 -22709.417} C_VEL
LIN {X 0,Y 190.313,Z 392.161,A -85,B 0,C 180,E1 -22711.054,E2 -22711.054} C_VEL
LIN {X 0,Y 191.779,Z 393.782,A -85,B 0,C 180,E1 -22711.888,E2 -22711.888} C_VEL
LIN {X 0,Y 194.707,Z 397.538,A -85,B 0,C 180,E1 -22713.495,E2 -22713.495} C_VEL
LIN {X 0,Y 199.471,Z 404.156,A -85,B 0,C 180,E1 -22715.911,E2 -22715.911} C_VEL
LIN {X 0,Y 204.02,Z 410.655,A -85,B 0,C 180,E1 -22718.006,E2 -22718.006} C_VEL
LIN {X 0,Y 205.522,Z 413.208,A -85,B 0,C 180,E1 -22718.68,E2 -22718.68} C_VEL
LIN {X 0,Y 206.957,Z 416.017,A -85,B 0,C 180,E1 -22719.325,E2 -22719.325} C_VEL
LIN {X 0,Y 208.033,Z 419.268,A -85,B 0,C 180,E1 -22719.857,E2 -22719.857} C_VEL
LIN {X 0,Y 209.489,Z 426.455,A -85,B 0,C 180,E1 -22720.704,E2 -22720.704} C_VEL
LIN {X 0,Y 210.763,Z 433.931,A -85,B 0,C 180,E1 -22721.483,E2 -22721.483} C_VEL
LIN {X 0,Y 212.187,Z 439.197,A -85,B 0,C 180,E1 -22722.178,E2 -22722.178} C_VEL
LIN {X 0,Y 212.836,Z 440.809,A -85,B 0,C 180,E1 -22722.449,E2 -22722.449} C_VEL
LIN {X 0,Y 215.588,Z 447.666,A -85,B 0,C 180,E1 -22723.569,E2 -22723.569} C_VEL
LIN {X 0,Y 212.075,Z 501.92,A -85,B 0,C 180,E1 -22725.16,E2 -22725.16} C_VEL
LIN {X 0,Y 210.624,Z 517.034,A -85,B 0,C 180,E1 -22725.77,E2 -22725.77} C_VEL
LIN {X 0,Y 208.41,Z 530.595,A -85,B 0,C 180,E1 -22726.604,E2 -22726.604} C_VEL
LIN {X 0,Y 205.338,Z 544.415,A -85,B 0,C 180,E1 -22727.806,E2 -22727.806} C_VEL
LIN {X 0,Y 201.978,Z 556.852,A -85,B 0,C 180,E1 -22729.279,E2 -22729.279} C_VEL
LIN {X 0,Y 198.249,Z 568.461,A -85,B 0,C 180,E1 -22731.048,E2 -22731.048} C_VEL
LIN {X 0,Y 194.489,Z 578.957,A -85,B 0,C 180,E1 -22733.08,E2 -22733.08} C_VEL
LIN {X 0,Y 189.915,Z 589.731,A -85,B 0,C 180,E1 -22735.647,E2 -22735.647} C_VEL
LIN {X 0,Y 185.435,Z 599.436,A -85,B 0,C 180,E1 -22738.596,E2 -22738.596} C_VEL
LIN {X 0,Y 181.441,Z 607.486,A -85,B 0,C 180,E1 -22741.677,E2 -22741.677} C_VEL
LIN {X 0,Y 177.621,Z 615.033,A -85,B 0,C 180,E1 -22745.352,E2 -22745.352} C_VEL
LIN {X 0,Y 174.834,Z 620.579,A -85,B 0,C 180,E1 -22748.794,E2 -22748.794} C_VEL
LIN {X 0,Y 172.585,Z 625,A -85,B 0,C 180,E1 -22752.22,E2 -22752.22} C_VEL
LIN {X 0,Y 170.903,Z 628.481,A -85,B 0,C 180,E1 -22755.719,E2 -22755.719} C_VEL
LIN {X 0,Y 169.476,Z 631.859,A -85,B 0,C 180,E1 -22760.455,E2 -22760.455} C_VEL
LIN {X 0,Y 168.93,Z 633.849,A -85,B 0,C 180,E1 -22765.23,E2 -22765.23} C_VEL
LIN {X 0,Y 168.849,Z 634.5,A -85,B 0,C 180,E1 -22770.003,E2 -22770.003} C_VEL
LIN {X 0,Y 168.937,Z 633.823,A -85,B 0,C 180,E1 -22774.776,E2 -22774.776} C_VEL
LIN {X 0,Y 169.671,Z 631.81,A -85,B 0,C 180,E1 -22779.54,E2 -22779.54} C_VEL
LIN {X 0,Y 170.964,Z 629.577,A -85,B 0,C 180,E1 -22783.07,E2 -22783.07} C_VEL
LIN {X 0,Y 172.656,Z 631.52,A -85,B 0,C 180,E1 -22786.558,E2 -22786.558} C_VEL
LIN {X 0,Y 176.026,Z 633.016,A -85,B 0,C 180,E1 -22791.062,E2 -22791.062} C_VEL
LIN {X 0,Y 180.695,Z 633.237,A -85,B 0,C 180,E1 -22795.333,E2 -22795.333} C_VEL
LIN {X 0,Y 186.605,Z 632.187,A -85,B 0,C 180,E1 -22799.318,E2 -22799.318} C_VEL
LIN {X 0,Y 193.737,Z 629.819,A -85,B 0,C 180,E1 -22802.969,E2 -22802.969} C_VEL
LIN {X 0,Y 201.848,Z 626.135,A -85,B 0,C 180,E1 -22806.295,E2 -22806.295} C_VEL
LIN {X 0,Y 208.495,Z 622.494,A -85,B 0,C 180,E1 -22808.582,E2 -22808.582} C_VEL
LIN {X 0,Y 218.205,Z 616.215,A -85,B 0,C 180,E1 -22811.323,E2 -22811.323} C_VEL
LIN {X 0,Y 227.265,Z 609.38,A -85,B 0,C 180,E1 -22813.48,E2 -22813.48} C_VEL
LIN {X 0,Y 236.801,Z 601.039,A -85,B 0,C 180,E1 -22815.424,E2 -22815.424} C_VEL
LIN {X 0,Y 236.43,Z 601.438,A -85,B 0,C 180,E1 -22815.812,E2 -22815.812} C_VEL
LIN {X 0,Y 227.101,Z 609.831,A -85,B 0,C 180,E1 -22817.694,E2 -22817.694} C_VEL
LIN {X 0,Y 217.973,Z 616.871,A -85,B 0,C 180,E1 -22819.846,E2 -22819.846} C_VEL
LIN {X 0,Y 208.342,Z 623.22,A -85,B 0,C 180,E1 -22822.613,E2 -22822.613} C_VEL
LIN {X 0,Y 199.461,Z 627.936,A -85,B 0,C 180,E1 -22825.684,E2 -22825.684} C_VEL
LIN {X 0,Y 191.564,Z 631.205,A -85,B 0,C 180,E1 -22829.094,E2 -22829.094} C_VEL
LIN {X 0,Y 187.933,Z 632.345,A -85,B 0,C 180,E1 -22830.912,E2 -22830.912} C_VEL
LIN {X 0,Y 184.655,Z 633.121,A -85,B 0,C 180,E1 -22832.824,E2 -22832.824} C_VEL
LIN {X 0,Y 179.21,Z 633.653,A -85,B 0,C 180,E1 -22836.911,E2 -22836.911} C_VEL
LIN {X 0,Y 174.988,Z 632.878,A -85,B 0,C 180,E1 -22841.259,E2 -22841.259} C_VEL
LIN {X 0,Y 171.95,Z 630.78,A -85,B 0,C 180,E1 -22845.804,E2 -22845.804} C_VEL
LIN {X 0,Y 170.261,Z 627.304,A -85,B 0,C 180,E1 -22850.496,E2 -22850.496} C_VEL
LIN {X 0,Y 169.846,Z 622.232,A -85,B 0,C 180,E1 -22855.253,E2 -22855.253} C_VEL
LIN {X 0,Y 170.05,Z 617.241,A -85,B 0,C 180,E1 -22858.816,E2 -22858.816} C_VEL
LIN {X 0,Y 170.346,Z 610.923,A -85,B 0,C 180,E1 -22862.365,E2 -22862.365} C_VEL
LIN {X 0,Y 170.574,Z 602.965,A -85,B 0,C 180,E1 -22865.912,E2 -22865.912} C_VEL
LIN {X 0,Y 171.026,Z 593.552,A -85,B 0,C 180,E1 -22869.254,E2 -22869.254} C_VEL
LIN {X 0,Y 171.761,Z 582.638,A -85,B 0,C 180,E1 -22872.405,E2 -22872.405} C_VEL
LIN {X 0,Y 172.643,Z 571.179,A -85,B 0,C 180,E1 -22875.042,E2 -22875.042} C_VEL
LIN {X 0,Y 173.642,Z 558.535,A -85,B 0,C 180,E1 -22877.368,E2 -22877.368} C_VEL
LIN {X 0,Y 174.541,Z 545.384,A -85,B 0,C 180,E1 -22879.249,E2 -22879.249} C_VEL
LIN {X 0,Y 175.458,Z 531.137,A -85,B 0,C 180,E1 -22880.747,E2 -22880.747} C_VEL
LIN {X 0,Y 177.126,Z 493.67,A -85,B 0,C 180,E1 -22883.62,E2 -22883.62} C_VEL
LIN {X 0,Y 178.903,Z 459.328,A -85,B 0,C 180,E1 -22886.15,E2 -22886.15} C_VEL
LIN {X 0,Y 177.712,Z 445.497,A -85,B 0,C 180,E1 -22887.291,E2 -22887.291} C_VEL
LIN {X 0,Y 177.693,Z 442.264,A -85,B 0,C 180,E1 -22887.853,E2 -22887.853} C_VEL
LIN {X 0,Y 178.016,Z 441.313,A -85,B 0,C 180,E1 -22888.279,E2 -22888.279} C_VEL
LIN {X 0,Y 179.339,Z 439.972,A -85,B 0,C 180,E1 -22889.013,E2 -22889.013} C_VEL
LIN {X 0,Y 181.227,Z 435.991,A -85,B 0,C 180,E1 -22889.763,E2 -22889.763} C_VEL
LIN {X 0,Y 183.777,Z 427.942,A -85,B 0,C 180,E1 -22890.524,E2 -22890.524} C_VEL
LIN {X 0,Y 184.671,Z 424.775,A -85,B 0,C 180,E1 -22890.757,E2 -22890.757} C_VEL
LIN {X 0,Y 187.004,Z 424.113,A -85,B 0,C 180,E1 -22891.892,E2 -22891.892} C_VEL
LIN {X 0,Y 190.273,Z 421.62,A -85,B 0,C 180,E1 -22893.274,E2 -22893.274} C_VEL
LIN {X 0,Y 191.718,Z 420.166,A -85,B 0,C 180,E1 -22893.831,E2 -22893.831} C_VEL
LIN {X 0,Y 194.594,Z 419.97,A -85,B 0,C 180,E1 -22895.063,E2 -22895.063} C_VEL
LIN {X 0,Y 197.122,Z 418.938,A -85,B 0,C 180,E1 -22896.035,E2 -22896.035} C_VEL
LIN {X 0,Y 201.923,Z 418.409,A -85,B 0,C 180,E1 -22897.839,E2 -22897.839} C_VEL
LIN {X 0,Y 208.457,Z 431.165,A -85,B 0,C 180,E1 -22900.761,E2 -22900.761} C_VEL
LIN {X 0,Y 213.38,Z 442.355,A -85,B 0,C 180,E1 -22902.818,E2 -22902.818} C_VEL
LIN {X 0,Y 215.365,Z 447.328,A -85,B 0,C 180,E1 -22903.622,E2 -22903.622} C_VEL
LIN {X 0,Y 212.24,Z 497.723,A -85,B 0,C 180,E1 -22905.137,E2 -22905.137} C_VEL
LIN {X 0,Y 210.811,Z 514.357,A -85,B 0,C 180,E1 -22905.729,E2 -22905.729} C_VEL
LIN {X 0,Y 208.743,Z 528.13,A -85,B 0,C 180,E1 -22906.518,E2 -22906.518} C_VEL
LIN {X 0,Y 205.882,Z 541.602,A -85,B 0,C 180,E1 -22907.606,E2 -22907.606} C_VEL
LIN {X 0,Y 202.514,Z 554.625,A -85,B 0,C 180,E1 -22909.075,E2 -22909.075} C_VEL
LIN {X 0,Y 198.442,Z 567.461,A -85,B 0,C 180,E1 -22910.967,E2 -22910.967} C_VEL
LIN {X 0,Y 194.092,Z 579.592,A -85,B 0,C 180,E1 -22913.309,E2 -22913.309} C_VEL
LIN {X 0,Y 189.963,Z 589.368,A -85,B 0,C 180,E1 -22915.651,E2 -22915.651} C_VEL
LIN {X 0,Y 185.476,Z 599.134,A -85,B 0,C 180,E1 -22918.597,E2 -22918.597} C_VEL
LIN {X 0,Y 181.489,Z 607.235,A -85,B 0,C 180,E1 -22921.679,E2 -22921.679} C_VEL
LIN {X 0,Y 177.502,Z 614.948,A -85,B 0,C 180,E1 -22925.402,E2 -22925.402} C_VEL
LIN {X 0,Y 174.84,Z 620.417,A -85,B 0,C 180,E1 -22928.788,E2 -22928.788} C_VEL
LIN {X 0,Y 172.597,Z 624.874,A -85,B 0,C 180,E1 -22932.215,E2 -22932.215} C_VEL
LIN {X 0,Y 170.918,Z 628.369,A -85,B 0,C 180,E1 -22935.714,E2 -22935.714} C_VEL
LIN {X 0,Y 169.481,Z 631.781,A -85,B 0,C 180,E1 -22940.449,E2 -22940.449} C_VEL
LIN {X 0,Y 168.933,Z 633.808,A -85,B 0,C 180,E1 -22945.224,E2 -22945.224} C_VEL
LIN {X 0,Y 168.85,Z 634.499,A -85,B 0,C 180,E1 -22949.997,E2 -22949.997} C_VEL
LIN {X 0,Y 168.931,Z 633.862,A -85,B 0,C 180,E1 -22954.77,E2 -22954.77} C_VEL
LIN {X 0,Y 169.476,Z 631.886,A -85,B 0,C 180,E1 -22959.545,E2 -22959.545} C_VEL
LIN {X 0,Y 170.898,Z 628.52,A -85,B 0,C 180,E1 -22964.282,E2 -22964.282} C_VEL
LIN {X 0,Y 173.274,Z 623.666,A -85,B 0,C 180,E1 -22968.931,E2 -22968.931} C_VEL
LIN {X 0,Y 176.536,Z 617.178,A -85,B 0,C 180,E1 -22973.456,E2 -22973.456} C_VEL
LIN {X 0,Y 180.195,Z 609.957,A -85,B 0,C 180,E1 -22977.272,E2 -22977.272} C_VEL
LIN {X 0,Y 184.657,Z 601.021,A -85,B 0,C 180,E1 -22980.914,E2 -22980.914} C_VEL
LIN {X 0,Y 189.047,Z 591.636,A -85,B 0,C 180,E1 -22983.889,E2 -22983.889} C_VEL
LIN {X 0,Y 193.518,Z 581.243,A -85,B 0,C 180,E1 -22986.487,E2 -22986.487} C_VEL
LIN {X 0,Y 197.654,Z 570.166,A -85,B 0,C 180,E1 -22988.705,E2 -22988.705} C_VEL
LIN {X 0,Y 201.452,Z 558.65,A -85,B 0,C 180,E1 -22990.52,E2 -22990.52} C_VEL
LIN {X 0,Y 204.804,Z 546.674,A -85,B 0,C 180,E1 -22991.998,E2 -22991.998} C_VEL
LIN {X 0,Y 207.773,Z 533.547,A -85,B 0,C 180,E1 -22993.229,E2 -22993.229} C_VEL
LIN {X 0,Y 210.235,Z 519.356,A -85,B 0,C 180,E1 -22994.166,E2 -22994.166} C_VEL
LIN {X 0,Y 211.873,Z 505.205,A -85,B 0,C 180,E1 -22994.763,E2 -22994.763} C_VEL
LIN {X 0,Y 215.538,Z 447.523,A -85,B 0,C 180,E1 -22996.497,E2 -22996.497} C_VEL
LIN {X 0,Y 209.795,Z 433.867,A -85,B 0,C 180,E1 -22998.865,E2 -22998.865} C_VEL
LIN {X 0,Y 204.194,Z 422.393,A -85,B 0,C 180,E1 -23001.324,E2 -23001.324} C_VEL
LIN {X 0,Y 199.854,Z 414.763,A -85,B 0,C 180,E1 -23003.353,E2 -23003.353} C_VEL
LIN {X 0,Y 194.508,Z 407.052,A -85,B 0,C 180,E1 -23006.019,E2 -23006.019} C_VEL
LIN {X 0,Y 191.473,Z 402.92,A -85,B 0,C 180,E1 -23007.672,E2 -23007.672} C_VEL
LIN {X 0,Y 188.333,Z 398.767,A -85,B 0,C 180,E1 -23009.517,E2 -23009.517} C_VEL
LIN {X 0,Y 185.561,Z 395.07,A -85,B 0,C 180,E1 -23011.293,E2 -23011.293} C_VEL
LIN {X 0,Y 184.697,Z 394.024,A -85,B 0,C 180,E1 -23011.87,E2 -23011.87} C_VEL
LIN {X 0,Y 181.977,Z 390.913,A -85,B 0,C 180,E1 -23013.786,E2 -23013.786} C_VEL
LIN {X 0,Y 180.838,Z 389.115,A -85,B 0,C 180,E1 -23014.691,E2 -23014.691} C_VEL
LIN {X 0,Y 178.193,Z 386.906,A -85,B 0,C 180,E1 -23016.771,E2 -23016.771} C_VEL
LIN {X 0,Y 176.386,Z 383.684,A -85,B 0,C 180,E1 -23018.526,E2 -23018.526} C_VEL
LIN {X 0,Y 173.573,Z 381.842,A -85,B 0,C 180,E1 -23021.253,E2 -23021.253} C_VEL
LIN {X 0,Y 171.952,Z 379.352,A -85,B 0,C 180,E1 -23023.299,E2 -23023.299} C_VEL
LIN {X 0,Y 171.661,Z 378.183,A -85,B 0,C 180,E1 -23024.262,E2 -23024.262} C_VEL
LIN {X 0,Y 171.604,Z 377.756,A -85,B 0,C 180,E1 -23025.775,E2 -23025.775} C_VEL
LIN {X 0,Y 171.882,Z 377.667,A -85,B 0,C 180,E1 -23030.587,E2 -23030.587} C_VEL
LIN {X 0,Y 171.815,Z 377.684,A -85,B 0,C 180,E1 -23035.307,E2 -23035.307} C_VEL
LIN {X 0,Y 172.328,Z 377.645,A -85,B 0,C 180,E1 -23040,E2 -23040} C_VEL
LIN {X 0,Y 171.815,Z 377.684,A -85,B 0,C 180,E1 -23044.692,E2 -23044.692} C_VEL
LIN {X 0,Y 171.882,Z 377.667,A -85,B 0,C 180,E1 -23049.413,E2 -23049.413} C_VEL
LIN {X 0,Y 171.588,Z 377.901,A -85,B 0,C 180,E1 -23055.136,E2 -23055.136} C_VEL
LIN {X 0,Y 171.818,Z 378.912,A -85,B 0,C 180,E1 -23056.485,E2 -23056.485} C_VEL
LIN {X 0,Y 173.169,Z 381.356,A -85,B 0,C 180,E1 -23058.332,E2 -23058.332} C_VEL
LIN {X 0,Y 175.605,Z 383.343,A -85,B 0,C 180,E1 -23060.824,E2 -23060.824} C_VEL
LIN {X 0,Y 176.615,Z 384.092,A -85,B 0,C 180,E1 -23061.751,E2 -23061.751} C_VEL
LIN {X 0,Y 178.251,Z 387.003,A -85,B 0,C 180,E1 -23063.327,E2 -23063.327} C_VEL
LIN {X 0,Y 181.23,Z 389.55,A -85,B 0,C 180,E1 -23065.654,E2 -23065.654} C_VEL
LIN {X 0,Y 183.481,Z 392.911,A -85,B 0,C 180,E1 -23067.364,E2 -23067.364} C_VEL
LIN {X 0,Y 185.536,Z 395.03,A -85,B 0,C 180,E1 -23068.735,E2 -23068.735} C_VEL
LIN {X 0,Y 188.375,Z 398.807,A -85,B 0,C 180,E1 -23070.552,E2 -23070.552} C_VEL
LIN {X 0,Y 193.167,Z 405.196,A -85,B 0,C 180,E1 -23073.309,E2 -23073.309} C_VEL
LIN {X 0,Y 198.188,Z 412.206,A -85,B 0,C 180,E1 -23075.886,E2 -23075.886} C_VEL
LIN {X 0,Y 202.013,Z 418.347,A -85,B 0,C 180,E1 -23077.712,E2 -23077.712} C_VEL
LIN {X 0,Y 208.018,Z 430.045,A -85,B 0,C 180,E1 -23080.418,E2 -23080.418} C_VEL
LIN {X 0,Y 212.836,Z 440.809,A -85,B 0,C 180,E1 -23082.449,E2 -23082.449} C_VEL
LIN {X 0,Y 213.441,Z 443.668,A -85,B 0,C 180,E1 -23082.765,E2 -23082.765} C_VEL
LIN {X 0,Y 213.058,Z 448.191,A -85,B 0,C 180,E1 -23082.874,E2 -23082.874} C_VEL
LIN {X 0,Y 210.097,Z 459.768,A -85,B 0,C 180,E1 -23082.573,E2 -23082.573} C_VEL
LIN {X 0,Y 209.842,Z 461.89,A -85,B 0,C 180,E1 -23082.602,E2 -23082.602} C_VEL
LIN {X 0,Y 206.423,Z 510.247,A -85,B 0,C 180,E1 -23084.079,E2 -23084.079} C_VEL
LIN {X 0,Y 204.407,Z 524.795,A -85,B 0,C 180,E1 -23084.839,E2 -23084.839} C_VEL
LIN {X 0,Y 201.733,Z 538.009,A -85,B 0,C 180,E1 -23085.836,E2 -23085.836} C_VEL
LIN {X 0,Y 198.102,Z 551.883,A -85,B 0,C 180,E1 -23087.278,E2 -23087.278} C_VEL
LIN {X 0,Y 194.23,Z 564.297,A -85,B 0,C 180,E1 -23089.021,E2 -23089.021} C_VEL
LIN {X 0,Y 190.079,Z 575.64,A -85,B 0,C 180,E1 -23091.06,E2 -23091.06} C_VEL
LIN {X 0,Y 186.617,Z 584.119,A -85,B 0,C 180,E1 -23092.95,E2 -23092.95} C_VEL
LIN {X 0,Y 181.653,Z 594.818,A -85,B 0,C 180,E1 -23095.879,E2 -23095.879} C_VEL
LIN {X 0,Y 177.23,Z 603.648,A -85,B 0,C 180,E1 -23098.972,E2 -23098.972} C_VEL
LIN {X 0,Y 172.695,Z 612.11,A -85,B 0,C 180,E1 -23102.756,E2 -23102.756} C_VEL
LIN {X 0,Y 169.125,Z 618.922,A -85,B 0,C 180,E1 -23106.752,E2 -23106.752} C_VEL
LIN {X 0,Y 166.577,Z 623.615,A -85,B 0,C 180,E1 -23110.277,E2 -23110.277} C_VEL
LIN {X 0,Y 163.976,Z 628.482,A -85,B 0,C 180,E1 -23115.102,E2 -23115.102} C_VEL
LIN {X 0,Y 162.449,Z 631.859,A -85,B 0,C 180,E1 -23120.038,E2 -23120.038} C_VEL
LIN {X 0,Y 161.85,Z 633.849,A -85,B 0,C 180,E1 -23125.021,E2 -23125.021} C_VEL
LIN {X 0,Y 161.772,Z 634.5,A -85,B 0,C 180,E1 -23130.003,E2 -23130.003} C_VEL
LIN {X 0,Y 161.859,Z 633.823,A -85,B 0,C 180,E1 -23134.985,E2 -23134.985} C_VEL
LIN {X 0,Y 162.681,Z 631.807,A -85,B 0,C 180,E1 -23139.954,E2 -23139.954} C_VEL
LIN {X 0,Y 164.439,Z 629.072,A -85,B 0,C 180,E1 -23144.387,E2 -23144.387} C_VEL
LIN {X 0,Y 167.425,Z 631.886,A -85,B 0,C 180,E1 -23149.625,E2 -23149.625} C_VEL
LIN {X 0,Y 171.749,Z 633.178,A -85,B 0,C 180,E1 -23154.158,E2 -23154.158} C_VEL
LIN {X 0,Y 177.211,Z 633.202,A -85,B 0,C 180,E1 -23158.421,E2 -23158.421} C_VEL
LIN {X 0,Y 184.049,Z 631.964,A -85,B 0,C 180,E1 -23162.32,E2 -23162.32} C_VEL
LIN {X 0,Y 191.982,Z 629.471,A -85,B 0,C 180,E1 -23165.857,E2 -23165.857} C_VEL
LIN {X 0,Y 200.836,Z 625.706,A -85,B 0,C 180,E1 -23169.045,E2 -23169.045} C_VEL
LIN {X 0,Y 210.627,Z 620.518,A -85,B 0,C 180,E1 -23171.865,E2 -23171.865} C_VEL
LIN {X 0,Y 221.126,Z 613.759,A -85,B 0,C 180,E1 -23174.367,E2 -23174.367} C_VEL
LIN {X 0,Y 226.625,Z 609.791,A -85,B 0,C 180,E1 -23175.504,E2 -23175.504} C_VEL
LIN {X 0,Y 223.57,Z 612.152,A -85,B 0,C 180,E1 -23176.245,E2 -23176.245} C_VEL
LIN {X 0,Y 215.427,Z 617.87,A -85,B 0,C 180,E1 -23178.027,E2 -23178.027} C_VEL
LIN {X 0,Y 205.322,Z 623.888,A -85,B 0,C 180,E1 -23180.711,E2 -23180.711} C_VEL
LIN {X 0,Y 198.195,Z 627.417,A -85,B 0,C 180,E1 -23182.928,E2 -23182.928} C_VEL
LIN {X 0,Y 189.497,Z 630.818,A -85,B 0,C 180,E1 -23186.199,E2 -23186.199} C_VEL
LIN {X 0,Y 181.797,Z 632.885,A -85,B 0,C 180,E1 -23189.831,E2 -23189.831} C_VEL
LIN {X 0,Y 178.376,Z 633.427,A -85,B 0,C 180,E1 -23191.784,E2 -23191.784} C_VEL
LIN {X 0,Y 172.7,Z 633.533,A -85,B 0,C 180,E1 -23195.987,E2 -23195.987} C_VEL
LIN {X 0,Y 168.302,Z 632.343,A -85,B 0,C 180,E1 -23200.484,E2 -23200.484} C_VEL
LIN {X 0,Y 165.144,Z 629.824,A -85,B 0,C 180,E1 -23205.206,E2 -23205.206} C_VEL
LIN {X 0,Y 163.41,Z 625.945,A -85,B 0,C 180,E1 -23210.094,E2 -23210.094} C_VEL
LIN {X 0,Y 162.954,Z 621.605,A -85,B 0,C 180,E1 -23214.172,E2 -23214.172} C_VEL
LIN {X 0,Y 163.145,Z 617.112,A -85,B 0,C 180,E1 -23217.531,E2 -23217.531} C_VEL
LIN {X 0,Y 163.403,Z 610.917,A -85,B 0,C 180,E1 -23221.232,E2 -23221.232} C_VEL
LIN {X 0,Y 163.677,Z 603.071,A -85,B 0,C 180,E1 -23224.927,E2 -23224.927} C_VEL
LIN {X 0,Y 164.034,Z 593.765,A -85,B 0,C 180,E1 -23228.427,E2 -23228.427} C_VEL
LIN {X 0,Y 164.681,Z 583.054,A -85,B 0,C 180,E1 -23231.695,E2 -23231.695} C_VEL
LIN {X 0,Y 165.546,Z 571.825,A -85,B 0,C 180,E1 -23234.443,E2 -23234.443} C_VEL
LIN {X 0,Y 166.503,Z 559.509,A -85,B 0,C 180,E1 -23236.87,E2 -23236.87} C_VEL
LIN {X 0,Y 167.423,Z 546.703,A -85,B 0,C 180,E1 -23238.827,E2 -23238.827} C_VEL
LIN {X 0,Y 168.257,Z 533.086,A -85,B 0,C 180,E1 -23240.397,E2 -23240.397} C_VEL
LIN {X 0,Y 169.299,Z 510.859,A -85,B 0,C 180,E1 -23242.26,E2 -23242.26} C_VEL
LIN {X 0,Y 171.208,Z 472.708,A -85,B 0,C 180,E1 -23245.342,E2 -23245.342} C_VEL
LIN {X 0,Y 171.597,Z 467.482,A -85,B 0,C 180,E1 -23246.026,E2 -23246.026} C_VEL
LIN {X 0,Y 172.076,Z 465.204,A -85,B 0,C 180,E1 -23246.572,E2 -23246.572} C_VEL
LIN {X 0,Y 173.377,Z 463.405,A -85,B 0,C 180,E1 -23247.377,E2 -23247.377} C_VEL
LIN {X 0,Y 175.964,Z 457.573,A -85,B 0,C 180,E1 -23248.478,E2 -23248.478} C_VEL
LIN {X 0,Y 179.112,Z 447.473,A -85,B 0,C 180,E1 -23249.486,E2 -23249.486} C_VEL
LIN {X 0,Y 181.313,Z 444.914,A -85,B 0,C 180,E1 -23250.5,E2 -23250.5} C_VEL
LIN {X 0,Y 183.584,Z 440.491,A -85,B 0,C 180,E1 -23251.359,E2 -23251.359} C_VEL
LIN {X 0,Y 186.181,Z 433.05,A -85,B 0,C 180,E1 -23252.123,E2 -23252.123} C_VEL
LIN {X 0,Y 186.811,Z 431.133,A -85,B 0,C 180,E1 -23252.295,E2 -23252.295} C_VEL
LIN {X 0,Y 190.477,Z 428.745,A -85,B 0,C 180,E1 -23253.843,E2 -23253.843} C_VEL
LIN {X 0,Y 192.224,Z 427.324,A -85,B 0,C 180,E1 -23254.521,E2 -23254.521} C_VEL
LIN {X 0,Y 195.859,Z 426.458,A -85,B 0,C 180,E1 -23255.986,E2 -23255.986} C_VEL
LIN {X 0,Y 197.468,Z 425.95,A -85,B 0,C 180,E1 -23256.594,E2 -23256.594} C_VEL
LIN {X 0,Y 199.718,Z 425.919,A -85,B 0,C 180,E1 -23257.454,E2 -23257.454} C_VEL
LIN {X 0,Y 205.557,Z 437.982,A -85,B 0,C 180,E1 -23260.176,E2 -23260.176} C_VEL
LIN {X 0,Y 210.39,Z 449.673,A -85,B 0,C 180,E1 -23262.296,E2 -23262.296} C_VEL
LIN {X 0,Y 206.617,Z 506.554,A -85,B 0,C 180,E1 -23264.034,E2 -23264.034} C_VEL
LIN {X 0,Y 204.853,Z 521.057,A -85,B 0,C 180,E1 -23264.696,E2 -23264.696} C_VEL
LIN {X 0,Y 202.292,Z 534.76,A -85,B 0,C 180,E1 -23265.636,E2 -23265.636} C_VEL
LIN {X 0,Y 199.233,Z 547.591,A -85,B 0,C 180,E1 -23266.882,E2 -23266.882} C_VEL
LIN {X 0,Y 195.247,Z 560.864,A -85,B 0,C 180,E1 -23268.589,E2 -23268.589} C_VEL
LIN {X 0,Y 191.171,Z 572.461,A -85,B 0,C 180,E1 -23270.536,E2 -23270.536} C_VEL
LIN {X 0,Y 186.673,Z 583.723,A -85,B 0,C 180,E1 -23272.957,E2 -23272.957} C_VEL
LIN {X 0,Y 181.69,Z 594.487,A -85,B 0,C 180,E1 -23275.88,E2 -23275.88} C_VEL
LIN {X 0,Y 177.28,Z 603.373,A -85,B 0,C 180,E1 -23278.975,E2 -23278.975} C_VEL
LIN {X 0,Y 172.746,Z 611.882,A -85,B 0,C 180,E1 -23282.758,E2 -23282.758} C_VEL
LIN {X 0,Y 169.987,Z 616.931,A -85,B 0,C 180,E1 -23285.576,E2 -23285.576} C_VEL
LIN {X 0,Y 166.59,Z 623.472,A -85,B 0,C 180,E1 -23290.272,E2 -23290.272} C_VEL
LIN {X 0,Y 163.992,Z 628.37,A -85,B 0,C 180,E1 -23295.097,E2 -23295.097} C_VEL
LIN {X 0,Y 162.454,Z 631.781,A -85,B 0,C 180,E1 -23300.032,E2 -23300.032} C_VEL
LIN {X 0,Y 161.852,Z 633.808,A -85,B 0,C 180,E1 -23305.015,E2 -23305.015} C_VEL
LIN {X 0,Y 161.774,Z 634.499,A -85,B 0,C 180,E1 -23309.997,E2 -23309.997} C_VEL
LIN {X 0,Y 161.851,Z 633.862,A -85,B 0,C 180,E1 -23314.979,E2 -23314.979} C_VEL
LIN {X 0,Y 162.449,Z 631.885,A -85,B 0,C 180,E1 -23319.962,E2 -23319.962} C_VEL
LIN {X 0,Y 163.971,Z 628.519,A -85,B 0,C 180,E1 -23324.899,E2 -23324.899} C_VEL
LIN {X 0,Y 166.55,Z 623.665,A -85,B 0,C 180,E1 -23329.726,E2 -23329.726} C_VEL
LIN {X 0,Y 169.998,Z 617.177,A -85,B 0,C 180,E1 -23334.416,E2 -23334.416} C_VEL
LIN {X 0,Y 173.881,Z 609.955,A -85,B 0,C 180,E1 -23338.35,E2 -23338.35} C_VEL
LIN {X 0,Y 178.589,Z 601.019,A -85,B 0,C 180,E1 -23342.087,E2 -23342.087} C_VEL
LIN {X 0,Y 183.193,Z 591.634,A -85,B 0,C 180,E1 -23345.128,E2 -23345.128} C_VEL
LIN {X 0,Y 188.227,Z 580.263,A -85,B 0,C 180,E1 -23347.997,E2 -23347.997} C_VEL
LIN {X 0,Y 192.738,Z 568.486,A -85,B 0,C 180,E1 -23350.329,E2 -23350.329} C_VEL
LIN {X 0,Y 196.587,Z 557.064,A -85,B 0,C 180,E1 -23352.087,E2 -23352.087} C_VEL
LIN {X 0,Y 200.084,Z 544.679,A -85,B 0,C 180,E1 -23353.573,E2 -23353.573} C_VEL
LIN {X 0,Y 203.186,Z 530.938,A -85,B 0,C 180,E1 -23354.805,E2 -23354.805} C_VEL
LIN {X 0,Y 205.641,Z 516.601,A -85,B 0,C 180,E1 -23355.685,E2 -23355.685} C_VEL
LIN {X 0,Y 207.145,Z 502.392,A -85,B 0,C 180,E1 -23356.235,E2 -23356.235} C_VEL
LIN {X 0,Y 210.557,Z 449.932,A -85,B 0,C 180,E1 -23357.823,E2 -23357.823} C_VEL
LIN {X 0,Y 205.725,Z 438.205,A -85,B 0,C 180,E1 -23359.948,E2 -23359.948} C_VEL
LIN {X 0,Y 200.338,Z 426.788,A -85,B 0,C 180,E1 -23362.469,E2 -23362.469} C_VEL
LIN {X 0,Y 196.344,Z 419.782,A -85,B 0,C 180,E1 -23364.441,E2 -23364.441} C_VEL
LIN {X 0,Y 191.436,Z 412.549,A -85,B 0,C 180,E1 -23367.034,E2 -23367.034} C_VEL
LIN {X 0,Y 188.544,Z 408.546,A -85,B 0,C 180,E1 -23368.7,E2 -23368.7} C_VEL
LIN {X 0,Y 185.725,Z 404.689,A -85,B 0,C 180,E1 -23370.454,E2 -23370.454} C_VEL
LIN {X 0,Y 182.524,Z 400.382,A -85,B 0,C 180,E1 -23372.635,E2 -23372.635} C_VEL
LIN {X 0,Y 179.704,Z 396.9,A -85,B 0,C 180,E1 -23374.743,E2 -23374.743} C_VEL
LIN {X 0,Y 178.935,Z 395.743,A -85,B 0,C 180,E1 -23375.378,E2 -23375.378} C_VEL
LIN {X 0,Y 176.135,Z 393.07,A -85,B 0,C 180,E1 -23377.724,E2 -23377.724} C_VEL
LIN {X 0,Y 174.691,Z 390.428,A -85,B 0,C 180,E1 -23379.206,E2 -23379.206} C_VEL
LIN {X 0,Y 171.978,Z 388.394,A -85,B 0,C 180,E1 -23381.998,E2 -23381.998} C_VEL
LIN {X 0,Y 170.266,Z 385.59,A -85,B 0,C 180,E1 -23384.283,E2 -23384.283} C_VEL
LIN {X 0,Y 169.78,Z 384.776,A -85,B 0,C 180,E1 -23385.006,E2 -23385.006} C_VEL
LIN {X 0,Y 166.408,Z 382.21,A -85,B 0,C 180,E1 -23390.887,E2 -23390.887} C_VEL
LIN {X 0,Y 165.126,Z 379.152,A -85,B 0,C 180,E1 -23397.484,E2 -23397.484} C_VEL
LIN {X 0,Y 165.324,Z 378.801,A -85,B 0,C 180,E1 -23400,E2 -23400} C_VEL
LIN {X 0,Y 165.082,Z 379.345,A -85,B 0,C 180,E1 -23403.05,E2 -23403.05} C_VEL
LIN {X 0,Y 168.926,Z 384.328,A -85,B 0,C 180,E1 -23413.841,E2 -23413.841} C_VEL
LIN {X 0,Y 170.15,Z 385.278,A -85,B 0,C 180,E1 -23415.574,E2 -23415.574} C_VEL
LIN {X 0,Y 171.707,Z 388.064,A -85,B 0,C 180,E1 -23417.723,E2 -23417.723} C_VEL
LIN {X 0,Y 174.237,Z 390.2,A -85,B 0,C 180,E1 -23420.416,E2 -23420.416} C_VEL
LIN {X 0,Y 174.89,Z 390.856,A -85,B 0,C 180,E1 -23421.058,E2 -23421.058} C_VEL
LIN {X 0,Y 176.68,Z 393.768,A -85,B 0,C 180,E1 -23422.82,E2 -23422.82} C_VEL
LIN {X 0,Y 179.348,Z 396.298,A -85,B 0,C 180,E1 -23425.005,E2 -23425.005} C_VEL
LIN {X 0,Y 182.105,Z 399.999,A -85,B 0,C 180,E1 -23427.122,E2 -23427.122} C_VEL
LIN {X 0,Y 183.208,Z 401.224,A -85,B 0,C 180,E1 -23427.889,E2 -23427.889} C_VEL
LIN {X 0,Y 186.353,Z 405.357,A -85,B 0,C 180,E1 -23429.98,E2 -23429.98} C_VEL
LIN {X 0,Y 192.72,Z 414.233,A -85,B 0,C 180,E1 -23433.706,E2 -23433.706} C_VEL
LIN {X 0,Y 197.848,Z 422.208,A -85,B 0,C 180,E1 -23436.354,E2 -23436.354} C_VEL
LIN {X 0,Y 203.524,Z 433.268,A -85,B 0,C 180,E1 -23439.085,E2 -23439.085} C_VEL
LIN {X 0,Y 209.048,Z 445.997,A -85,B 0,C 180,E1 -23441.565,E2 -23441.565} C_VEL
LIN {X 0,Y 210.595,Z 450.005,A -85,B 0,C 180,E1 -23442.237,E2 -23442.237} C_VEL
LIN {X 0,Y 209.842,Z 461.89,A -85,B 0,C 180,E1 -23442.602,E2 -23442.602} C_VEL
LIN {X 0,Y 208.989,Z 467.743,A -85,B 0,C 180,E1 -23442.639,E2 -23442.639} C_VEL
LIN {X 0,Y 203.815,Z 486.791,A -85,B 0,C 180,E1 -23442.025,E2 -23442.025} C_VEL
LIN {X 0,Y 202.974,Z 492.644,A -85,B 0,C 180,E1 -23442.065,E2 -23442.065} C_VEL
LIN {X 0,Y 201.318,Z 512.303,A -85,B 0,C 180,E1 -23442.724,E2 -23442.724} C_VEL
LIN {X 0,Y 199.211,Z 526.327,A -85,B 0,C 180,E1 -23443.5,E2 -23443.5} C_VEL
LIN {X 0,Y 196.172,Z 540.275,A -85,B 0,C 180,E1 -23444.603,E2 -23444.603} C_VEL
LIN {X 0,Y 192.438,Z 553.655,A -85,B 0,C 180,E1 -23446.065,E2 -23446.065} C_VEL
LIN {X 0,Y 188.429,Z 565.719,A -85,B 0,C 180,E1 -23447.832,E2 -23447.832} C_VEL
LIN {X 0,Y 184.16,Z 576.812,A -85,B 0,C 180,E1 -23449.915,E2 -23449.915} C_VEL
LIN {X 0,Y 180.092,Z 586.072,A -85,B 0,C 180,E1 -23452.079,E2 -23452.079} C_VEL
LIN {X 0,Y 174.983,Z 596.446,A -85,B 0,C 180,E1 -23455.091,E2 -23455.091} C_VEL
LIN {X 0,Y 170.428,Z 605.003,A -85,B 0,C 180,E1 -23458.283,E2 -23458.283} C_VEL
LIN {X 0,Y 165.786,Z 613.189,A -85,B 0,C 180,E1 -23462.209,E2 -23462.209} C_VEL
LIN {X 0,Y 162.587,Z 618.924,A -85,B 0,C 180,E1 -23465.758,E2 -23465.758} C_VEL
LIN {X 0,Y 159.89,Z 623.616,A -85,B 0,C 180,E1 -23469.416,E2 -23469.416} C_VEL
LIN {X 0,Y 157.074,Z 628.483,A -85,B 0,C 180,E1 -23474.431,E2 -23474.431} C_VEL
LIN {X 0,Y 155.445,Z 631.86,A -85,B 0,C 180,E1 -23479.584,E2 -23479.584} C_VEL
LIN {X 0,Y 154.755,Z 633.85,A -85,B 0,C 180,E1 -23484.792,E2 -23484.792} C_VEL
LIN {X 0,Y 154.684,Z 634.5,A -85,B 0,C 180,E1 -23490.003,E2 -23490.003} C_VEL
LIN {X 0,Y 154.771,Z 633.822,A -85,B 0,C 180,E1 -23495.214,E2 -23495.214} C_VEL
LIN {X 0,Y 155.683,Z 631.807,A -85,B 0,C 180,E1 -23500.406,E2 -23500.406} C_VEL
LIN {X 0,Y 157.938,Z 628.453,A -85,B 0,C 180,E1 -23505.737,E2 -23505.737} C_VEL
LIN {X 0,Y 160.773,Z 631.203,A -85,B 0,C 180,E1 -23510.473,E2 -23510.473} C_VEL
LIN {X 0,Y 165.313,Z 632.885,A -85,B 0,C 180,E1 -23515.162,E2 -23515.162} C_VEL
LIN {X 0,Y 171.017,Z 633.346,A -85,B 0,C 180,E1 -23519.551,E2 -23519.551} C_VEL
LIN {X 0,Y 178.119,Z 632.605,A -85,B 0,C 180,E1 -23523.535,E2 -23523.535} C_VEL
LIN {X 0,Y 186.36,Z 630.647,A -85,B 0,C 180,E1 -23527.116,E2 -23527.116} C_VEL
LIN {X 0,Y 195.522,Z 627.456,A -85,B 0,C 180,E1 -23530.319,E2 -23530.319} C_VEL
LIN {X 0,Y 205.595,Z 622.919,A -85,B 0,C 180,E1 -23533.134,E2 -23533.134} C_VEL
LIN {X 0,Y 214.614,Z 617.98,A -85,B 0,C 180,E1 -23535.224,E2 -23535.224} C_VEL
LIN {X 0,Y 215.446,Z 617.489,A -85,B 0,C 180,E1 -23535.684,E2 -23535.684} C_VEL
LIN {X 0,Y 205.146,Z 623.354,A -85,B 0,C 180,E1 -23538.084,E2 -23538.084} C_VEL
LIN {X 0,Y 197.522,Z 626.939,A -85,B 0,C 180,E1 -23540.174,E2 -23540.174} C_VEL
LIN {X 0,Y 188.061,Z 630.482,A -85,B 0,C 180,E1 -23543.278,E2 -23543.278} C_VEL
LIN {X 0,Y 179.592,Z 632.668,A -85,B 0,C 180,E1 -23546.78,E2 -23546.78} C_VEL
LIN {X 0,Y 172.163,Z 633.575,A -85,B 0,C 180,E1 -23550.669,E2 -23550.669} C_VEL
LIN {X 0,Y 166.243,Z 633.22,A -85,B 0,C 180,E1 -23554.992,E2 -23554.992} C_VEL
LIN {X 0,Y 161.651,Z 631.63,A -85,B 0,C 180,E1 -23559.647,E2 -23559.647} C_VEL
LIN {X 0,Y 158.389,Z 628.726,A -85,B 0,C 180,E1 -23564.56,E2 -23564.56} C_VEL
LIN {X 0,Y 156.591,Z 624.449,A -85,B 0,C 180,E1 -23569.658,E2 -23569.658} C_VEL
LIN {X 0,Y 156.189,Z 618.642,A -85,B 0,C 180,E1 -23574.837,E2 -23574.837} C_VEL
LIN {X 0,Y 156.408,Z 612.985,A -85,B 0,C 180,E1 -23578.713,E2 -23578.713} C_VEL
LIN {X 0,Y 156.672,Z 607.16,A -85,B 0,C 180,E1 -23581.928,E2 -23581.928} C_VEL
LIN {X 0,Y 156.854,Z 600.087,A -85,B 0,C 180,E1 -23585.142,E2 -23585.142} C_VEL
LIN {X 0,Y 157.237,Z 591.083,A -85,B 0,C 180,E1 -23588.494,E2 -23588.494} C_VEL
LIN {X 0,Y 157.861,Z 580.792,A -85,B 0,C 180,E1 -23591.624,E2 -23591.624} C_VEL
LIN {X 0,Y 158.668,Z 569.535,A -85,B 0,C 180,E1 -23594.428,E2 -23594.428} C_VEL
LIN {X 0,Y 159.634,Z 556.634,A -85,B 0,C 180,E1 -23596.958,E2 -23596.958} C_VEL
LIN {X 0,Y 160.467,Z 544.327,A -85,B 0,C 180,E1 -23598.845,E2 -23598.845} C_VEL
LIN {X 0,Y 161.347,Z 530.077,A -85,B 0,C 180,E1 -23600.477,E2 -23600.477} C_VEL
LIN {X 0,Y 162.305,Z 508.853,A -85,B 0,C 180,E1 -23602.433,E2 -23602.433} C_VEL
LIN {X 0,Y 162.663,Z 504.024,A -85,B 0,C 180,E1 -23603.22,E2 -23603.22} C_VEL
LIN {X 0,Y 162.855,Z 502.992,A -85,B 0,C 180,E1 -23603.527,E2 -23603.527} C_VEL
LIN {X 0,Y 163.578,Z 502.049,A -85,B 0,C 180,E1 -23604.174,E2 -23604.174} C_VEL
LIN {X 0,Y 164.954,Z 499.414,A -85,B 0,C 180,E1 -23604.965,E2 -23604.965} C_VEL
LIN {X 0,Y 167.48,Z 491.93,A -85,B 0,C 180,E1 -23606.056,E2 -23606.056} C_VEL
LIN {X 0,Y 173.105,Z 471.512,A -85,B 0,C 180,E1 -23607.915,E2 -23607.915} C_VEL
LIN {X 0,Y 173.74,Z 470.422,A -85,B 0,C 180,E1 -23608.215,E2 -23608.215} C_VEL
LIN {X 0,Y 175.499,Z 467.856,A -85,B 0,C 180,E1 -23609.057,E2 -23609.057} C_VEL
LIN {X 0,Y 178.581,Z 461.154,A -85,B 0,C 180,E1 -23610.271,E2 -23610.271} C_VEL
LIN {X 0,Y 181.449,Z 452.412,A -85,B 0,C 180,E1 -23611.14,E2 -23611.14} C_VEL
LIN {X 0,Y 183.966,Z 449.003,A -85,B 0,C 180,E1 -23612.171,E2 -23612.171} C_VEL
LIN {X 0,Y 186.813,Z 443.239,A -85,B 0,C 180,E1 -23613.14,E2 -23613.14} C_VEL
LIN {X 0,Y 189.174,Z 436.801,A -85,B 0,C 180,E1 -23613.792,E2 -23613.792} C_VEL
LIN {X 0,Y 192.785,Z 434.211,A -85,B 0,C 180,E1 -23615.201,E2 -23615.201} C_VEL
LIN {X 0,Y 197.842,Z 434.228,A -85,B 0,C 180,E1 -23617.23,E2 -23617.23} C_VEL
LIN {X 0,Y 202.663,Z 444.869,A -85,B 0,C 180,E1 -23619.573,E2 -23619.573} C_VEL
LIN {X 0,Y 205.503,Z 452.099,A -85,B 0,C 180,E1 -23620.902,E2 -23620.902} C_VEL
LIN {X 0,Y 202.606,Z 495.422,A -85,B 0,C 180,E1 -23622.236,E2 -23622.236} C_VEL
LIN {X 0,Y 201.035,Z 513.247,A -85,B 0,C 180,E1 -23622.854,E2 -23622.854} C_VEL
LIN {X 0,Y 198.845,Z 527.388,A -85,B 0,C 180,E1 -23623.657,E2 -23623.657} C_VEL
LIN {X 0,Y 195.618,Z 541.616,A -85,B 0,C 180,E1 -23624.798,E2 -23624.798} C_VEL
LIN {X 0,Y 191.994,Z 554.636,A -85,B 0,C 180,E1 -23626.293,E2 -23626.293} C_VEL
LIN {X 0,Y 187.896,Z 566.63,A -85,B 0,C 180,E1 -23628.074,E2 -23628.074} C_VEL
LIN {X 0,Y 183.323,Z 578.53,A -85,B 0,C 180,E1 -23630.403,E2 -23630.403} C_VEL
LIN {X 0,Y 178.414,Z 589.374,A -85,B 0,C 180,E1 -23633.075,E2 -23633.075} C_VEL
LIN {X 0,Y 173.47,Z 599.139,A -85,B 0,C 180,E1 -23636.143,E2 -23636.143} C_VEL
LIN {X 0,Y 169.071,Z 607.239,A -85,B 0,C 180,E1 -23639.385,E2 -23639.385} C_VEL
LIN {X 0,Y 164.62,Z 614.998,A -85,B 0,C 180,E1 -23643.364,E2 -23643.364} C_VEL
LIN {X 0,Y 161.595,Z 620.419,A -85,B 0,C 180,E1 -23646.954,E2 -23646.954} C_VEL
LIN {X 0,Y 159.101,Z 624.876,A -85,B 0,C 180,E1 -23650.649,E2 -23650.649} C_VEL
LIN {X 0,Y 157.09,Z 628.371,A -85,B 0,C 180,E1 -23654.426,E2 -23654.426} C_VEL
LIN {X 0,Y 155.451,Z 631.782,A -85,B 0,C 180,E1 -23659.578,E2 -23659.578} C_VEL
LIN {X 0,Y 154.757,Z 633.808,A -85,B 0,C 180,E1 -23664.786,E2 -23664.786} C_VEL
LIN {X 0,Y 154.686,Z 634.499,A -85,B 0,C 180,E1 -23669.997,E2 -23669.997} C_VEL
LIN {X 0,Y 154.756,Z 633.862,A -85,B 0,C 180,E1 -23675.208,E2 -23675.208} C_VEL
LIN {X 0,Y 155.445,Z 631.885,A -85,B 0,C 180,E1 -23680.416,E2 -23680.416} C_VEL
LIN {X 0,Y 157.068,Z 628.519,A -85,B 0,C 180,E1 -23685.57,E2 -23685.57} C_VEL
LIN {X 0,Y 159.864,Z 623.663,A -85,B 0,C 180,E1 -23690.588,E2 -23690.588} C_VEL
LIN {X 0,Y 163.5,Z 617.175,A -85,B 0,C 180,E1 -23695.454,E2 -23695.454} C_VEL
LIN {X 0,Y 167.646,Z 609.953,A -85,B 0,C 180,E1 -23699.506,E2 -23699.506} C_VEL
LIN {X 0,Y 172.601,Z 601.017,A -85,B 0,C 180,E1 -23703.342,E2 -23703.342} C_VEL
LIN {X 0,Y 177.43,Z 591.631,A -85,B 0,C 180,E1 -23706.448,E2 -23706.448} C_VEL
LIN {X 0,Y 182.545,Z 580.566,A -85,B 0,C 180,E1 -23709.302,E2 -23709.302} C_VEL
LIN {X 0,Y 187.366,Z 568.482,A -85,B 0,C 180,E1 -23711.738,E2 -23711.738} C_VEL
LIN {X 0,Y 191.366,Z 557.058,A -85,B 0,C 180,E1 -23713.515,E2 -23713.515} C_VEL
LIN {X 0,Y 195.009,Z 544.672,A -85,B 0,C 180,E1 -23715.009,E2 -23715.009} C_VEL
LIN {X 0,Y 198.222,Z 530.93,A -85,B 0,C 180,E1 -23716.249,E2 -23716.249} C_VEL
LIN {X 0,Y 200.76,Z 516.589,A -85,B 0,C 180,E1 -23717.131,E2 -23717.131} C_VEL
LIN {X 0,Y 202.29,Z 502.708,A -85,B 0,C 180,E1 -23717.672,E2 -23717.672} C_VEL
LIN {X 0,Y 205.722,Z 452.411,A -85,B 0,C 180,E1 -23719.2,E2 -23719.2} C_VEL
LIN {X 0,Y 201.074,Z 440.937,A -85,B 0,C 180,E1 -23721.397,E2 -23721.397} C_VEL
LIN {X 0,Y 196.267,Z 430.783,A -85,B 0,C 180,E1 -23723.8,E2 -23723.8} C_VEL
LIN {X 0,Y 193.06,Z 424.979,A -85,B 0,C 180,E1 -23725.491,E2 -23725.491} C_VEL
LIN {X 0,Y 188.57,Z 418.211,A -85,B 0,C 180,E1 -23728,E2 -23728} C_VEL
LIN {X 0,Y 185.606,Z 414.032,A -85,B 0,C 180,E1 -23729.808,E2 -23729.808} C_VEL
LIN {X 0,Y 183.078,Z 410.475,A -85,B 0,C 180,E1 -23731.48,E2 -23731.48} C_VEL
LIN {X 0,Y 180.256,Z 406.55,A -85,B 0,C 180,E1 -23733.516,E2 -23733.516} C_VEL
LIN {X 0,Y 177.384,Z 402.761,A -85,B 0,C 180,E1 -23735.805,E2 -23735.805} C_VEL
LIN {X 0,Y 173.938,Z 398.93,A -85,B 0,C 180,E1 -23738.894,E2 -23738.894} C_VEL
LIN {X 0,Y 172.997,Z 397.123,A -85,B 0,C 180,E1 -23739.928,E2 -23739.928} C_VEL
LIN {X 0,Y 170.3,Z 394.795,A -85,B 0,C 180,E1 -23742.9,E2 -23742.9} C_VEL
LIN {X 0,Y 168.661,Z 391.831,A -85,B 0,C 180,E1 -23745.29,E2 -23745.29} C_VEL
LIN {X 0,Y 164.801,Z 388.299,A -85,B 0,C 180,E1 -23752.957,E2 -23752.957} C_VEL
LIN {X 0,Y 163.915,Z 386.028,A -85,B 0,C 180,E1 -23758.157,E2 -23758.157} C_VEL
LIN {X 0,Y 163.862,Z 385.757,A -85,B 0,C 180,E1 -23760,E2 -23760} C_VEL
LIN {X 0,Y 164.043,Z 386.567,A -85,B 0,C 180,E1 -23763.377,E2 -23763.377} C_VEL
LIN {X 0,Y 167.691,Z 391.225,A -85,B 0,C 180,E1 -23773.327,E2 -23773.327} C_VEL
LIN {X 0,Y 168.679,Z 391.875,A -85,B 0,C 180,E1 -23774.785,E2 -23774.785} C_VEL
LIN {X 0,Y 170.379,Z 394.904,A -85,B 0,C 180,E1 -23777.246,E2 -23777.246} C_VEL
LIN {X 0,Y 173.18,Z 397.51,A -85,B 0,C 180,E1 -23780.327,E2 -23780.327} C_VEL
LIN {X 0,Y 175.375,Z 400.812,A -85,B 0,C 180,E1 -23782.532,E2 -23782.532} C_VEL
LIN {X 0,Y 177.418,Z 402.844,A -85,B 0,C 180,E1 -23784.272,E2 -23784.272} C_VEL
LIN {X 0,Y 180.378,Z 406.708,A -85,B 0,C 180,E1 -23786.62,E2 -23786.62} C_VEL
LIN {X 0,Y 185.075,Z 413.248,A -85,B 0,C 180,E1 -23789.894,E2 -23789.894} C_VEL
LIN {X 0,Y 188.313,Z 417.821,A -85,B 0,C 180,E1 -23791.892,E2 -23791.892} C_VEL
LIN {X 0,Y 192.875,Z 424.722,A -85,B 0,C 180,E1 -23794.457,E2 -23794.457} C_VEL
LIN {X 0,Y 195.868,Z 430.034,A -85,B 0,C 180,E1 -23796.04,E2 -23796.04} C_VEL
LIN {X 0,Y 200.876,Z 440.45,A -85,B 0,C 180,E1 -23798.55,E2 -23798.55} C_VEL
LIN {X 0,Y 205.721,Z 452.313,A -85,B 0,C 180,E1 -23800.839,E2 -23800.839} C_VEL
LIN {X 0,Y 202.974,Z 492.644,A -85,B 0,C 180,E1 -23802.065,E2 -23802.065} C_VEL
LIN {X 0,Y 202.12,Z 498.497,A -85,B 0,C 180,E1 -23802.098,E2 -23802.098} C_VEL
LIN {X 0,Y 196.914,Z 515.505,A -85,B 0,C 180,E1 -23801.579,E2 -23801.579} C_VEL
LIN {X 0,Y 195.372,Z 521.199,A -85,B 0,C 180,E1 -23801.664,E2 -23801.664} C_VEL
LIN {X 0,Y 194.991,Z 523.098,A -85,B 0,C 180,E1 -23801.767,E2 -23801.767} C_VEL
LIN {X 0,Y 192.088,Z 536.893,A -85,B 0,C 180,E1 -23802.779,E2 -23802.779} C_VEL
LIN {X 0,Y 188.469,Z 550.127,A -85,B 0,C 180,E1 -23804.129,E2 -23804.129} C_VEL
LIN {X 0,Y 184.252,Z 562.881,A -85,B 0,C 180,E1 -23805.888,E2 -23805.888} C_VEL
LIN {X 0,Y 179.422,Z 575.148,A -85,B 0,C 180,E1 -23808.093,E2 -23808.093} C_VEL
LIN {X 0,Y 175.48,Z 584.125,A -85,B 0,C 180,E1 -23810.153,E2 -23810.153} C_VEL
LIN {X 0,Y 170.049,Z 594.823,A -85,B 0,C 180,E1 -23813.186,E2 -23813.186} C_VEL
LIN {X 0,Y 165.16,Z 603.652,A -85,B 0,C 180,E1 -23816.418,E2 -23816.418} C_VEL
LIN {X 0,Y 160.146,Z 612.113,A -85,B 0,C 180,E1 -23820.42,E2 -23820.42} C_VEL
LIN {X 0,Y 156.067,Z 618.979,A -85,B 0,C 180,E1 -23824.718,E2 -23824.718} C_VEL
LIN {X 0,Y 153.241,Z 623.617,A -85,B 0,C 180,E1 -23828.479,E2 -23828.479} C_VEL
LIN {X 0,Y 150.2,Z 628.483,A -85,B 0,C 180,E1 -23833.699,E2 -23833.699} C_VEL
LIN {X 0,Y 148.433,Z 631.86,A -85,B 0,C 180,E1 -23839.086,E2 -23839.086} C_VEL
LIN {X 0,Y 147.687,Z 633.85,A -85,B 0,C 180,E1 -23844.542,E2 -23844.542} C_VEL
LIN {X 0,Y 147.588,Z 634.5,A -85,B 0,C 180,E1 -23850.003,E2 -23850.003} C_VEL
LIN {X 0,Y 147.704,Z 633.822,A -85,B 0,C 180,E1 -23855.464,E2 -23855.464} C_VEL
LIN {X 0,Y 148.707,Z 631.806,A -85,B 0,C 180,E1 -23860.9,E2 -23860.9} C_VEL
LIN {X 0,Y 150.967,Z 628.428,A -85,B 0,C 180,E1 -23866.223,E2 -23866.223} C_VEL
LIN {X 0,Y 151.587,Z 627.78,A -85,B 0,C 180,E1 -23867.195,E2 -23867.195} C_VEL
LIN {X 0,Y 154.186,Z 630.298,A -85,B 0,C 180,E1 -23871.389,E2 -23871.389} C_VEL
LIN {X 0,Y 158.933,Z 632.407,A -85,B 0,C 180,E1 -23876.248,E2 -23876.248} C_VEL
LIN {X 0,Y 164.896,Z 633.322,A -85,B 0,C 180,E1 -23880.764,E2 -23880.764} C_VEL
LIN {X 0,Y 172.276,Z 633.068,A -85,B 0,C 180,E1 -23884.832,E2 -23884.832} C_VEL
LIN {X 0,Y 180.819,Z 631.627,A -85,B 0,C 180,E1 -23888.457,E2 -23888.457} C_VEL
LIN {X 0,Y 190.268,Z 628.997,A -85,B 0,C 180,E1 -23891.676,E2 -23891.676} C_VEL
LIN {X 0,Y 200.629,Z 625.084,A -85,B 0,C 180,E1 -23894.478,E2 -23894.478} C_VEL
LIN {X 0,Y 203.935,Z 623.62,A -85,B 0,C 180,E1 -23895.245,E2 -23895.245} C_VEL
LIN {X 0,Y 203.875,Z 623.675,A -85,B 0,C 180,E1 -23895.852,E2 -23895.852} C_VEL
LIN {X 0,Y 192.227,Z 628.533,A -85,B 0,C 180,E1 -23898.845,E2 -23898.845} C_VEL
LIN {X 0,Y 182.483,Z 631.507,A -85,B 0,C 180,E1 -23901.96,E2 -23901.96} C_VEL
LIN {X 0,Y 173.725,Z 633.156,A -85,B 0,C 180,E1 -23905.503,E2 -23905.503} C_VEL
LIN {X 0,Y 166.023,Z 633.559,A -85,B 0,C 180,E1 -23909.471,E2 -23909.471} C_VEL
LIN {X 0,Y 159.848,Z 632.748,A -85,B 0,C 180,E1 -23913.917,E2 -23913.917} C_VEL
LIN {X 0,Y 155.069,Z 630.734,A -85,B 0,C 180,E1 -23918.742,E2 -23918.742} C_VEL
LIN {X 0,Y 151.677,Z 627.449,A -85,B 0,C 180,E1 -23923.859,E2 -23923.859} C_VEL
LIN {X 0,Y 149.824,Z 622.761,A -85,B 0,C 180,E1 -23929.185,E2 -23929.185} C_VEL
LIN {X 0,Y 149.446,Z 616.538,A -85,B 0,C 180,E1 -23934.603,E2 -23934.603} C_VEL
LIN {X 0,Y 149.659,Z 610.542,A -85,B 0,C 180,E1 -23938.655,E2 -23938.655} C_VEL
LIN {X 0,Y 149.926,Z 604.357,A -85,B 0,C 180,E1 -23942.015,E2 -23942.015} C_VEL
LIN {X 0,Y 150.158,Z 596.818,A -85,B 0,C 180,E1 -23945.371,E2 -23945.371} C_VEL
LIN {X 0,Y 150.504,Z 586.855,A -85,B 0,C 180,E1 -23949.002,E2 -23949.002} C_VEL
LIN {X 0,Y 151.197,Z 575.68,A -85,B 0,C 180,E1 -23952.278,E2 -23952.278} C_VEL
LIN {X 0,Y 152.086,Z 563.874,A -85,B 0,C 180,E1 -23955.066,E2 -23955.066} C_VEL
LIN {X 0,Y 153.126,Z 549.559,A -85,B 0,C 180,E1 -23957.702,E2 -23957.702} C_VEL
LIN {X 0,Y 154.008,Z 535.25,A -85,B 0,C 180,E1 -23959.667,E2 -23959.667} C_VEL
LIN {X 0,Y 154.27,Z 529.963,A -85,B 0,C 180,E1 -23960.414,E2 -23960.414} C_VEL
LIN {X 0,Y 154.5,Z 527.71,A -85,B 0,C 180,E1 -23961.079,E2 -23961.079} C_VEL
LIN {X 0,Y 155.246,Z 527.079,A -85,B 0,C 180,E1 -23961.931,E2 -23961.931} C_VEL
LIN {X 0,Y 156.696,Z 525.394,A -85,B 0,C 180,E1 -23962.758,E2 -23962.758} C_VEL
LIN {X 0,Y 158.896,Z 521.379,A -85,B 0,C 180,E1 -23963.624,E2 -23963.624} C_VEL
LIN {X 0,Y 163.302,Z 509.821,A -85,B 0,C 180,E1 -23964.954,E2 -23964.954} C_VEL
LIN {X 0,Y 163.817,Z 508.74,A -85,B 0,C 180,E1 -23965.176,E2 -23965.176} C_VEL
LIN {X 0,Y 165.855,Z 505.788,A -85,B 0,C 180,E1 -23966.302,E2 -23966.302} C_VEL
LIN {X 0,Y 167.856,Z 501.381,A -85,B 0,C 180,E1 -23967.198,E2 -23967.198} C_VEL
LIN {X 0,Y 170.444,Z 493.689,A -85,B 0,C 180,E1 -23968.181,E2 -23968.181} C_VEL
LIN {X 0,Y 175.528,Z 475.714,A -85,B 0,C 180,E1 -23969.716,E2 -23969.716} C_VEL
LIN {X 0,Y 177.94,Z 471.986,A -85,B 0,C 180,E1 -23970.764,E2 -23970.764} C_VEL
LIN {X 0,Y 181.231,Z 465.071,A -85,B 0,C 180,E1 -23971.967,E2 -23971.967} C_VEL
LIN {X 0,Y 184.13,Z 456.865,A -85,B 0,C 180,E1 -23972.811,E2 -23972.811} C_VEL
LIN {X 0,Y 187.021,Z 452.546,A -85,B 0,C 180,E1 -23973.871,E2 -23973.871} C_VEL
LIN {X 0,Y 190.05,Z 446.379,A -85,B 0,C 180,E1 -23974.812,E2 -23974.812} C_VEL
LIN {X 0,Y 191.801,Z 442.125,A -85,B 0,C 180,E1 -23975.288,E2 -23975.288} C_VEL
LIN {X 0,Y 193.37,Z 441.129,A -85,B 0,C 180,E1 -23975.878,E2 -23975.878} C_VEL
LIN {X 0,Y 195.302,Z 441.288,A -85,B 0,C 180,E1 -23976.665,E2 -23976.665} C_VEL
LIN {X 0,Y 199.904,Z 452.162,A -85,B 0,C 180,E1 -23979.016,E2 -23979.016} C_VEL
LIN {X 0,Y 200.8,Z 454.459,A -85,B 0,C 180,E1 -23979.457,E2 -23979.457} C_VEL
LIN {X 0,Y 196.75,Z 509.631,A -85,B 0,C 180,E1 -23981.184,E2 -23981.184} C_VEL
LIN {X 0,Y 194.58,Z 524.35,A -85,B 0,C 180,E1 -23981.939,E2 -23981.939} C_VEL
LIN {X 0,Y 191.559,Z 538.246,A -85,B 0,C 180,E1 -23982.986,E2 -23982.986} C_VEL
LIN {X 0,Y 188.027,Z 551.176,A -85,B 0,C 180,E1 -23984.366,E2 -23984.366} C_VEL
LIN {X 0,Y 183.775,Z 563.724,A -85,B 0,C 180,E1 -23986.117,E2 -23986.117} C_VEL
LIN {X 0,Y 179.303,Z 575.172,A -85,B 0,C 180,E1 -23988.212,E2 -23988.212} C_VEL
LIN {X 0,Y 174.591,Z 585.679,A -85,B 0,C 180,E1 -23990.651,E2 -23990.651} C_VEL
LIN {X 0,Y 169.235,Z 596.119,A -85,B 0,C 180,E1 -23993.714,E2 -23993.714} C_VEL
LIN {X 0,Y 164.449,Z 604.731,A -85,B 0,C 180,E1 -23996.979,E2 -23996.979} C_VEL
LIN {X 0,Y 159.546,Z 612.984,A -85,B 0,C 180,E1 -24001.014,E2 -24001.014} C_VEL
LIN {X 0,Y 155.936,Z 618.953,A -85,B 0,C 180,E1 -24004.812,E2 -24004.812} C_VEL
LIN {X 0,Y 152.379,Z 624.877,A -85,B 0,C 180,E1 -24009.759,E2 -24009.759} C_VEL
LIN {X 0,Y 150.216,Z 628.372,A -85,B 0,C 180,E1 -24013.694,E2 -24013.694} C_VEL
LIN {X 0,Y 148.439,Z 631.783,A -85,B 0,C 180,E1 -24019.08,E2 -24019.08} C_VEL
LIN {X 0,Y 147.69,Z 633.809,A -85,B 0,C 180,E1 -24024.535,E2 -24024.535} C_VEL
LIN {X 0,Y 147.589,Z 634.499,A -85,B 0,C 180,E1 -24029.997,E2 -24029.997} C_VEL
LIN {X 0,Y 147.688,Z 633.862,A -85,B 0,C 180,E1 -24035.458,E2 -24035.458} C_VEL
LIN {X 0,Y 148.433,Z 631.884,A -85,B 0,C 180,E1 -24040.914,E2 -24040.914} C_VEL
LIN {X 0,Y 150.194,Z 628.518,A -85,B 0,C 180,E1 -24046.302,E2 -24046.302} C_VEL
LIN {X 0,Y 153.215,Z 623.662,A -85,B 0,C 180,E1 -24051.525,E2 -24051.525} C_VEL
LIN {X 0,Y 157.072,Z 617.174,A -85,B 0,C 180,E1 -24056.576,E2 -24056.576} C_VEL
LIN {X 0,Y 161.472,Z 609.951,A -85,B 0,C 180,E1 -24060.754,E2 -24060.754} C_VEL
LIN {X 0,Y 166.687,Z 601.014,A -85,B 0,C 180,E1 -24064.69,E2 -24064.69} C_VEL
LIN {X 0,Y 171.753,Z 591.628,A -85,B 0,C 180,E1 -24067.86,E2 -24067.86} C_VEL
LIN {X 0,Y 176.927,Z 580.934,A -85,B 0,C 180,E1 -24070.677,E2 -24070.677} C_VEL
LIN {X 0,Y 181.631,Z 569.766,A -85,B 0,C 180,E1 -24072.994,E2 -24072.994} C_VEL
LIN {X 0,Y 186.283,Z 557.053,A -85,B 0,C 180,E1 -24075.019,E2 -24075.019} C_VEL
LIN {X 0,Y 190.05,Z 544.665,A -85,B 0,C 180,E1 -24076.525,E2 -24076.525} C_VEL
LIN {X 0,Y 193.387,Z 530.921,A -85,B 0,C 180,E1 -24077.766,E2 -24077.766} C_VEL
LIN {X 0,Y 196.01,Z 516.577,A -85,B 0,C 180,E1 -24078.648,E2 -24078.648} C_VEL
LIN {X 0,Y 197.608,Z 502.229,A -85,B 0,C 180,E1 -24079.211,E2 -24079.211} C_VEL
LIN {X 0,Y 200.967,Z 454.701,A -85,B 0,C 180,E1 -24080.669,E2 -24080.669} C_VEL
LIN {X 0,Y 196.147,Z 442.751,A -85,B 0,C 180,E1 -24083.127,E2 -24083.127} C_VEL
LIN {X 0,Y 191.188,Z 432.437,A -85,B 0,C 180,E1 -24085.824,E2 -24085.824} C_VEL
LIN {X 0,Y 186.309,Z 424.677,A -85,B 0,C 180,E1 -24088.657,E2 -24088.657} C_VEL
LIN {X 0,Y 182.886,Z 419.669,A -85,B 0,C 180,E1 -24090.857,E2 -24090.857} C_VEL
LIN {X 0,Y 180.136,Z 415.804,A -85,B 0,C 180,E1 -24092.793,E2 -24092.793} C_VEL
LIN {X 0,Y 178.196,Z 412.953,A -85,B 0,C 180,E1 -24094.288,E2 -24094.288} C_VEL
LIN {X 0,Y 174.846,Z 408.539,A -85,B 0,C 180,E1 -24097.122,E2 -24097.122} C_VEL
LIN {X 0,Y 172.175,Z 405.34,A -85,B 0,C 180,E1 -24099.7,E2 -24099.7} C_VEL
LIN {X 0,Y 171.177,Z 403.705,A -85,B 0,C 180,E1 -24100.825,E2 -24100.825} C_VEL
LIN {X 0,Y 168.454,Z 400.932,A -85,B 0,C 180,E1 -24104.11,E2 -24104.11} C_VEL
LIN {X 0,Y 167.267,Z 398.511,A -85,B 0,C 180,E1 -24106.019,E2 -24106.019} C_VEL
LIN {X 0,Y 163.949,Z 395.515,A -85,B 0,C 180,E1 -24112.843,E2 -24112.843} C_VEL
LIN {X 0,Y 163.046,Z 393.109,A -85,B 0,C 180,E1 -24118.147,E2 -24118.147} C_VEL
LIN {X 0,Y 162.999,Z 392.786,A -85,B 0,C 180,E1 -24120,E2 -24120} C_VEL
LIN {X 0,Y 163.169,Z 393.7,A -85,B 0,C 180,E1 -24123.395,E2 -24123.395} C_VEL
LIN {X 0,Y 166.844,Z 398.312,A -85,B 0,C 180,E1 -24133.396,E2 -24133.396} C_VEL
LIN {X 0,Y 167.409,Z 398.855,A -85,B 0,C 180,E1 -24134.279,E2 -24134.279} C_VEL
LIN {X 0,Y 169.173,Z 401.887,A -85,B 0,C 180,E1 -24136.906,E2 -24136.906} C_VEL
LIN {X 0,Y 171.538,Z 404.19,A -85,B 0,C 180,E1 -24139.622,E2 -24139.622} C_VEL
LIN {X 0,Y 173.965,Z 407.72,A -85,B 0,C 180,E1 -24142.138,E2 -24142.138} C_VEL
LIN {X 0,Y 175.602,Z 409.456,A -85,B 0,C 180,E1 -24143.592,E2 -24143.592} C_VEL
LIN {X 0,Y 178.491,Z 413.252,A -85,B 0,C 180,E1 -24145.979,E2 -24145.979} C_VEL
LIN {X 0,Y 182.805,Z 419.563,A -85,B 0,C 180,E1 -24149.135,E2 -24149.135} C_VEL
LIN {X 0,Y 187.131,Z 425.828,A -85,B 0,C 180,E1 -24151.88,E2 -24151.88} C_VEL
LIN {X 0,Y 191.74,Z 433.49,A -85,B 0,C 180,E1 -24154.531,E2 -24154.531} C_VEL
LIN {X 0,Y 196.848,Z 444.425,A -85,B 0,C 180,E1 -24157.288,E2 -24157.288} C_VEL
LIN {X 0,Y 200.97,Z 454.708,A -85,B 0,C 180,E1 -24159.378,E2 -24159.378} C_VEL
LIN {X 0,Y 197.854,Z 498.331,A -85,B 0,C 180,E1 -24160.705,E2 -24160.705} C_VEL
LIN {X 0,Y 196.387,Z 513.966,A -85,B 0,C 180,E1 -24161.283,E2 -24161.283} C_VEL
LIN {X 0,Y 194.991,Z 523.098,A -85,B 0,C 180,E1 -24161.767,E2 -24161.767} C_VEL
LIN {X 0,Y 193.456,Z 528.745,A -85,B 0,C 180,E1 -24161.982,E2 -24161.982} C_VEL
LIN {X 0,Y 189.405,Z 537.816,A -85,B 0,C 180,E1 -24162.056,E2 -24162.056} C_VEL
LIN {X 0,Y 185.065,Z 546.743,A -85,B 0,C 180,E1 -24162.293,E2 -24162.293} C_VEL
LIN {X 0,Y 183.003,Z 552.002,A -85,B 0,C 180,E1 -24162.766,E2 -24162.766} C_VEL
LIN {X 0,Y 178.683,Z 564.31,A -85,B 0,C 180,E1 -24164.534,E2 -24164.534} C_VEL
LIN {X 0,Y 173.519,Z 576.783,A -85,B 0,C 180,E1 -24166.876,E2 -24166.876} C_VEL
LIN {X 0,Y 169.109,Z 586.078,A -85,B 0,C 180,E1 -24169.119,E2 -24169.119} C_VEL
LIN {X 0,Y 163.52,Z 596.451,A -85,B 0,C 180,E1 -24172.237,E2 -24172.237} C_VEL
LIN {X 0,Y 158.483,Z 605.007,A -85,B 0,C 180,E1 -24175.574,E2 -24175.574} C_VEL
LIN {X 0,Y 153.29,Z 613.192,A -85,B 0,C 180,E1 -24179.718,E2 -24179.718} C_VEL
LIN {X 0,Y 149.254,Z 619.572,A -85,B 0,C 180,E1 -24183.992,E2 -24183.992} C_VEL
LIN {X 0,Y 145.694,Z 625.003,A -85,B 0,C 180,E1 -24188.794,E2 -24188.794} C_VEL
LIN {X 0,Y 143.359,Z 628.484,A -85,B 0,C 180,E1 -24192.898,E2 -24192.898} C_VEL
LIN {X 0,Y 141.441,Z 631.861,A -85,B 0,C 180,E1 -24198.54,E2 -24198.54} C_VEL
LIN {X 0,Y 140.619,Z 633.85,A -85,B 0,C 180,E1 -24204.267,E2 -24204.267} C_VEL
LIN {X 0,Y 140.502,Z 634.5,A -85,B 0,C 180,E1 -24210.004,E2 -24210.004} C_VEL
LIN {X 0,Y 140.637,Z 633.822,A -85,B 0,C 180,E1 -24215.74,E2 -24215.74} C_VEL
LIN {X 0,Y 141.728,Z 631.806,A -85,B 0,C 180,E1 -24221.444,E2 -24221.444} C_VEL
LIN {X 0,Y 144.163,Z 628.409,A -85,B 0,C 180,E1 -24227.011,E2 -24227.011} C_VEL
LIN {X 0,Y 145.441,Z 627.061,A -85,B 0,C 180,E1 -24228.949,E2 -24228.949} C_VEL
LIN {X 0,Y 149.961,Z 630.635,A -85,B 0,C 180,E1 -24234.951,E2 -24234.951} C_VEL
LIN {X 0,Y 155.505,Z 632.57,A -85,B 0,C 180,E1 -24239.815,E2 -24239.815} C_VEL
LIN {X 0,Y 162.508,Z 633.373,A -85,B 0,C 180,E1 -24244.212,E2 -24244.212} C_VEL
LIN {X 0,Y 170.801,Z 633.029,A -85,B 0,C 180,E1 -24248.116,E2 -24248.116} C_VEL
LIN {X 0,Y 180.112,Z 631.531,A -85,B 0,C 180,E1 -24251.559,E2 -24251.559} C_VEL
LIN {X 0,Y 190.344,Z 628.851,A -85,B 0,C 180,E1 -24254.553,E2 -24254.553} C_VEL
LIN {X 0,Y 193.133,Z 627.936,A -85,B 0,C 180,E1 -24255.266,E2 -24255.266} C_VEL
LIN {X 0,Y 192.328,Z 628.236,A -85,B 0,C 180,E1 -24256.029,E2 -24256.029} C_VEL
LIN {X 0,Y 181.879,Z 631.287,A -85,B 0,C 180,E1 -24258.936,E2 -24258.936} C_VEL
LIN {X 0,Y 172.297,Z 633.05,A -85,B 0,C 180,E1 -24262.277,E2 -24262.277} C_VEL
LIN {X 0,Y 163.771,Z 633.563,A -85,B 0,C 180,E1 -24266.091,E2 -24266.091} C_VEL
LIN {X 0,Y 159.963,Z 633.364,A -85,B 0,C 180,E1 -24268.182,E2 -24268.182} C_VEL
LIN {X 0,Y 153.527,Z 632.095,A -85,B 0,C 180,E1 -24272.757,E2 -24272.757} C_VEL
LIN {X 0,Y 148.547,Z 629.651,A -85,B 0,C 180,E1 -24277.76,E2 -24277.76} C_VEL
LIN {X 0,Y 145.019,Z 625.958,A -85,B 0,C 180,E1 -24283.096,E2 -24283.096} C_VEL
LIN {X 0,Y 143.107,Z 620.922,A -85,B 0,C 180,E1 -24288.671,E2 -24288.671} C_VEL
LIN {X 0,Y 142.753,Z 614.265,A -85,B 0,C 180,E1 -24294.35,E2 -24294.35} C_VEL
LIN {X 0,Y 142.989,Z 607.876,A -85,B 0,C 180,E1 -24298.592,E2 -24298.592} C_VEL
LIN {X 0,Y 143.196,Z 601.301,A -85,B 0,C 180,E1 -24302.11,E2 -24302.11} C_VEL
LIN {X 0,Y 143.41,Z 593.269,A -85,B 0,C 180,E1 -24305.625,E2 -24305.625} C_VEL
LIN {X 0,Y 143.79,Z 583.409,A -85,B 0,C 180,E1 -24309.154,E2 -24309.154} C_VEL
LIN {X 0,Y 144.521,Z 571.968,A -85,B 0,C 180,E1 -24312.484,E2 -24312.484} C_VEL
LIN {X 0,Y 145.394,Z 559.352,A -85,B 0,C 180,E1 -24315.417,E2 -24315.417} C_VEL
LIN {X 0,Y 146.309,Z 545.243,A -85,B 0,C 180,E1 -24318.013,E2 -24318.013} C_VEL
LIN {X 0,Y 146.386,Z 543.336,A -85,B 0,C 180,E1 -24318.728,E2 -24318.728} C_VEL
LIN {X 0,Y 146.568,Z 542.953,A -85,B 0,C 180,E1 -24319.248,E2 -24319.248} C_VEL
LIN {X 0,Y 146.81,Z 542.92,A -85,B 0,C 180,E1 -24319.579,E2 -24319.579} C_VEL
LIN {X 0,Y 148.474,Z 541.696,A -85,B 0,C 180,E1 -24320.794,E2 -24320.794} C_VEL
LIN {X 0,Y 151.016,Z 538.243,A -85,B 0,C 180,E1 -24321.858,E2 -24321.858} C_VEL
LIN {X 0,Y 153.35,Z 534.285,A -85,B 0,C 180,E1 -24322.534,E2 -24322.534} C_VEL
LIN {X 0,Y 155.82,Z 532.035,A -85,B 0,C 180,E1 -24323.95,E2 -24323.95} C_VEL
LIN {X 0,Y 158.081,Z 529.204,A -85,B 0,C 180,E1 -24324.927,E2 -24324.927} C_VEL
LIN {X 0,Y 161.026,Z 523.996,A -85,B 0,C 180,E1 -24325.878,E2 -24325.878} C_VEL
LIN {X 0,Y 165.402,Z 513.547,A -85,B 0,C 180,E1 -24327.017,E2 -24327.017} C_VEL
LIN {X 0,Y 167.656,Z 510.359,A -85,B 0,C 180,E1 -24328.053,E2 -24328.053} C_VEL
LIN {X 0,Y 169.951,Z 505.765,A -85,B 0,C 180,E1 -24328.971,E2 -24328.971} C_VEL
LIN {X 0,Y 172.793,Z 498.14,A -85,B 0,C 180,E1 -24329.968,E2 -24329.968} C_VEL
LIN {X 0,Y 177.769,Z 480.981,A -85,B 0,C 180,E1 -24331.363,E2 -24331.363} C_VEL
LIN {X 0,Y 178.372,Z 479.624,A -85,B 0,C 180,E1 -24331.577,E2 -24331.577} C_VEL
LIN {X 0,Y 181.402,Z 474.482,A -85,B 0,C 180,E1 -24332.735,E2 -24332.735} C_VEL
LIN {X 0,Y 184.522,Z 467.795,A -85,B 0,C 180,E1 -24333.758,E2 -24333.758} C_VEL
LIN {X 0,Y 187.076,Z 460.995,A -85,B 0,C 180,E1 -24334.462,E2 -24334.462} C_VEL
LIN {X 0,Y 190.369,Z 455.816,A -85,B 0,C 180,E1 -24335.554,E2 -24335.554} C_VEL
LIN {X 0,Y 193.411,Z 449.86,A -85,B 0,C 180,E1 -24336.434,E2 -24336.434} C_VEL
LIN {X 0,Y 196.173,Z 456.91,A -85,B 0,C 180,E1 -24337.927,E2 -24337.927} C_VEL
LIN {X 0,Y 192.106,Z 510.06,A -85,B 0,C 180,E1 -24339.611,E2 -24339.611} C_VEL
LIN {X 0,Y 189.923,Z 524.36,A -85,B 0,C 180,E1 -24340.35,E2 -24340.35} C_VEL
LIN {X 0,Y 186.796,Z 538.253,A -85,B 0,C 180,E1 -24341.395,E2 -24341.395} C_VEL
LIN {X 0,Y 183.134,Z 551.182,A -85,B 0,C 180,E1 -24342.778,E2 -24342.778} C_VEL
LIN {X 0,Y 178.717,Z 563.729,A -85,B 0,C 180,E1 -24344.536,E2 -24344.536} C_VEL
LIN {X 0,Y 174.04,Z 575.175,A -85,B 0,C 180,E1 -24346.644,E2 -24346.644} C_VEL
LIN {X 0,Y 169.15,Z 585.682,A -85,B 0,C 180,E1 -24349.123,E2 -24349.123} C_VEL
LIN {X 0,Y 163.561,Z 596.121,A -85,B 0,C 180,E1 -24352.24,E2 -24352.24} C_VEL
LIN {X 0,Y 158.519,Z 604.733,A -85,B 0,C 180,E1 -24355.575,E2 -24355.575} C_VEL
LIN {X 0,Y 153.335,Z 612.985,A -85,B 0,C 180,E1 -24359.72,E2 -24359.72} C_VEL
LIN {X 0,Y 149.699,Z 618.553,A -85,B 0,C 180,E1 -24363.35,E2 -24363.35} C_VEL
LIN {X 0,Y 146.624,Z 623.475,A -85,B 0,C 180,E1 -24367.448,E2 -24367.448} C_VEL
LIN {X 0,Y 143.375,Z 628.373,A -85,B 0,C 180,E1 -24372.892,E2 -24372.892} C_VEL
LIN {X 0,Y 141.447,Z 631.783,A -85,B 0,C 180,E1 -24378.533,E2 -24378.533} C_VEL
LIN {X 0,Y 140.622,Z 633.809,A -85,B 0,C 180,E1 -24384.26,E2 -24384.26} C_VEL
LIN {X 0,Y 140.503,Z 634.499,A -85,B 0,C 180,E1 -24389.996,E2 -24389.996} C_VEL
LIN {X 0,Y 140.62,Z 633.861,A -85,B 0,C 180,E1 -24395.733,E2 -24395.733} C_VEL
LIN {X 0,Y 141.44,Z 631.884,A -85,B 0,C 180,E1 -24401.46,E2 -24401.46} C_VEL
LIN {X 0,Y 143.353,Z 628.517,A -85,B 0,C 180,E1 -24407.103,E2 -24407.103} C_VEL
LIN {X 0,Y 146.588,Z 623.661,A -85,B 0,C 180,E1 -24412.55,E2 -24412.55} C_VEL
LIN {X 0,Y 150.719,Z 617.172,A -85,B 0,C 180,E1 -24417.79,E2 -24417.79} C_VEL
LIN {X 0,Y 155.389,Z 609.949,A -85,B 0,C 180,E1 -24422.098,E2 -24422.098} C_VEL
LIN {X 0,Y 160.854,Z 601.012,A -85,B 0,C 180,E1 -24426.141,E2 -24426.141} C_VEL
LIN {X 0,Y 166.177,Z 591.625,A -85,B 0,C 180,E1 -24429.37,E2 -24429.37} C_VEL
LIN {X 0,Y 171.439,Z 581.262,A -85,B 0,C 180,E1 -24432.149,E2 -24432.149} C_VEL
LIN {X 0,Y 176.489,Z 569.762,A -85,B 0,C 180,E1 -24434.571,E2 -24434.571} C_VEL
LIN {X 0,Y 181.34,Z 557.048,A -85,B 0,C 180,E1 -24436.604,E2 -24436.604} C_VEL
LIN {X 0,Y 185.227,Z 544.659,A -85,B 0,C 180,E1 -24438.122,E2 -24438.122} C_VEL
LIN {X 0,Y 188.684,Z 530.913,A -85,B 0,C 180,E1 -24439.364,E2 -24439.364} C_VEL
LIN {X 0,Y 191.396,Z 516.565,A -85,B 0,C 180,E1 -24440.243,E2 -24440.243} C_VEL
LIN {X 0,Y 193.024,Z 502.467,A -85,B 0,C 180,E1 -24440.798,E2 -24440.798} C_VEL
LIN {X 0,Y 196.366,Z 457.194,A -85,B 0,C 180,E1 -24442.19,E2 -24442.19} C_VEL
LIN {X 0,Y 191.711,Z 445.541,A -85,B 0,C 180,E1 -24444.753,E2 -24444.753} C_VEL
LIN {X 0,Y 187.577,Z 436.916,A -85,B 0,C 180,E1 -24447.172,E2 -24447.172} C_VEL
LIN {X 0,Y 182.903,Z 429.363,A -85,B 0,C 180,E1 -24450.091,E2 -24450.091} C_VEL
LIN {X 0,Y 178.565,Z 422.862,A -85,B 0,C 180,E1 -24453.167,E2 -24453.167} C_VEL
LIN {X 0,Y 175.847,Z 418.947,A -85,B 0,C 180,E1 -24455.345,E2 -24455.345} C_VEL
LIN {X 0,Y 173.056,Z 415.063,A -85,B 0,C 180,E1 -24457.854,E2 -24457.854} C_VEL
LIN {X 0,Y 170.353,Z 411.628,A -85,B 0,C 180,E1 -24460.627,E2 -24460.627} C_VEL
LIN {X 0,Y 169.552,Z 410.372,A -85,B 0,C 180,E1 -24461.575,E2 -24461.575} C_VEL
LIN {X 0,Y 166.879,Z 407.318,A -85,B 0,C 180,E1 -24465.051,E2 -24465.051} C_VEL
LIN {X 0,Y 165.838,Z 405.288,A -85,B 0,C 180,E1 -24466.833,E2 -24466.833} C_VEL
LIN {X 0,Y 162.594,Z 401.727,A -85,B 0,C 180,E1 -24474.73,E2 -24474.73} C_VEL
LIN {X 0,Y 162.147,Z 400.044,A -85,B 0,C 180,E1 -24478.758,E2 -24478.758} C_VEL
LIN {X 0,Y 162.146,Z 400.033,A -85,B 0,C 180,E1 -24481.242,E2 -24481.242} C_VEL
LIN {X 0,Y 166.075,Z 405.614,A -85,B 0,C 180,E1 -24493.615,E2 -24493.615} C_VEL
LIN {X 0,Y 167.977,Z 408.834,A -85,B 0,C 180,E1 -24496.56,E2 -24496.56} C_VEL
LIN {X 0,Y 169.946,Z 410.868,A -85,B 0,C 180,E1 -24498.927,E2 -24498.927} C_VEL
LIN {X 0,Y 172.558,Z 414.599,A -85,B 0,C 180,E1 -24501.73,E2 -24501.73} C_VEL
LIN {X 0,Y 173.833,Z 416.118,A -85,B 0,C 180,E1 -24502.921,E2 -24502.921} C_VEL
LIN {X 0,Y 177.093,Z 420.702,A -85,B 0,C 180,E1 -24505.725,E2 -24505.725} C_VEL
LIN {X 0,Y 180.704,Z 426.047,A -85,B 0,C 180,E1 -24508.45,E2 -24508.45} C_VEL
LIN {X 0,Y 185.131,Z 432.836,A -85,B 0,C 180,E1 -24511.385,E2 -24511.385} C_VEL
LIN {X 0,Y 188.748,Z 439.174,A -85,B 0,C 180,E1 -24513.572,E2 -24513.572} C_VEL
LIN {X 0,Y 193.237,Z 449.113,A -85,B 0,C 180,E1 -24516.148,E2 -24516.148} C_VEL
LIN {X 0,Y 196.387,Z 457.304,A -85,B 0,C 180,E1 -24517.87,E2 -24517.87} C_VEL
LIN {X 0,Y 192.78,Z 504.596,A -85,B 0,C 180,E1 -24519.302,E2 -24519.302} C_VEL
LIN {X 0,Y 191.013,Z 518.908,A -85,B 0,C 180,E1 -24519.927,E2 -24519.927} C_VEL
LIN {X 0,Y 188.202,Z 533.227,A -85,B 0,C 180,E1 -24520.875,E2 -24520.875} C_VEL
LIN {X 0,Y 184.729,Z 546.427,A -85,B 0,C 180,E1 -24522.113,E2 -24522.113} C_VEL
LIN {X 0,Y 183.003,Z 552.002,A -85,B 0,C 180,E1 -24522.766,E2 -24522.766} C_VEL
LIN {X 0,Y 180.809,Z 557.242,A -85,B 0,C 180,E1 -24523.293,E2 -24523.293} C_VEL
LIN {X 0,Y 175.69,Z 565.57,A -85,B 0,C 180,E1 -24523.88,E2 -24523.88} C_VEL
LIN {X 0,Y 170.3,Z 573.524,A -85,B 0,C 180,E1 -24524.672,E2 -24524.672} C_VEL
LIN {X 0,Y 167.715,Z 578.171,A -85,B 0,C 180,E1 -24525.532,E2 -24525.532} C_VEL
LIN {X 0,Y 162.787,Z 587.963,A -85,B 0,C 180,E1 -24528.001,E2 -24528.001} C_VEL
LIN {X 0,Y 156.991,Z 597.962,A -85,B 0,C 180,E1 -24531.195,E2 -24531.195} C_VEL
LIN {X 0,Y 151.823,Z 606.265,A -85,B 0,C 180,E1 -24534.65,E2 -24534.65} C_VEL
LIN {X 0,Y 146.465,Z 614.201,A -85,B 0,C 180,E1 -24538.951,E2 -24538.951} C_VEL
LIN {X 0,Y 142.157,Z 620.585,A -85,B 0,C 180,E1 -24543.585,E2 -24543.585} C_VEL
LIN {X 0,Y 138.151,Z 626.246,A -85,B 0,C 180,E1 -24549.143,E2 -24549.143} C_VEL
LIN {X 0,Y 135.376,Z 630.352,A -85,B 0,C 180,E1 -24554.959,E2 -24554.959} C_VEL
LIN {X 0,Y 133.855,Z 633.025,A -85,B 0,C 180,E1 -24560.941,E2 -24560.941} C_VEL
LIN {X 0,Y 133.397,Z 634.341,A -85,B 0,C 180,E1 -24566.984,E2 -24566.984} C_VEL
LIN {X 0,Y 133.418,Z 634.5,A -85,B 0,C 180,E1 -24570.004,E2 -24570.004} C_VEL
LIN {X 0,Y 133.566,Z 633.821,A -85,B 0,C 180,E1 -24576.045,E2 -24576.045} C_VEL
LIN {X 0,Y 134.774,Z 631.805,A -85,B 0,C 180,E1 -24582.043,E2 -24582.043} C_VEL
LIN {X 0,Y 137.395,Z 628.408,A -85,B 0,C 180,E1 -24587.877,E2 -24587.877} C_VEL
LIN {X 0,Y 139.488,Z 626.258,A -85,B 0,C 180,E1 -24590.849,E2 -24590.849} C_VEL
LIN {X 0,Y 143.619,Z 629.587,A -85,B 0,C 180,E1 -24596.134,E2 -24596.134} C_VEL
LIN {X 0,Y 149.407,Z 631.942,A -85,B 0,C 180,E1 -24601.164,E2 -24601.164} C_VEL
LIN {X 0,Y 156.7,Z 633.202,A -85,B 0,C 180,E1 -24605.669,E2 -24605.669} C_VEL
LIN {X 0,Y 165.285,Z 633.356,A -85,B 0,C 180,E1 -24609.632,E2 -24609.632} C_VEL
LIN {X 0,Y 174.901,Z 632.388,A -85,B 0,C 180,E1 -24613.09,E2 -24613.09} C_VEL
LIN {X 0,Y 182.432,Z 630.958,A -85,B 0,C 180,E1 -24615.287,E2 -24615.287} C_VEL
LIN {X 0,Y 181.885,Z 631.102,A -85,B 0,C 180,E1 -24615.932,E2 -24615.932} C_VEL
LIN {X 0,Y 171.558,Z 632.939,A -85,B 0,C 180,E1 -24619.046,E2 -24619.046} C_VEL
LIN {X 0,Y 162.236,Z 633.554,A -85,B 0,C 180,E1 -24622.665,E2 -24622.665} C_VEL
LIN {X 0,Y 153.993,Z 632.976,A -85,B 0,C 180,E1 -24626.793,E2 -24626.793} C_VEL
LIN {X 0,Y 147.293,Z 631.265,A -85,B 0,C 180,E1 -24631.501,E2 -24631.501} C_VEL
LIN {X 0,Y 142.111,Z 628.403,A -85,B 0,C 180,E1 -24636.695,E2 -24636.695} C_VEL
LIN {X 0,Y 138.447,Z 624.287,A -85,B 0,C 180,E1 -24642.267,E2 -24642.267} C_VEL
LIN {X 0,Y 136.466,Z 618.826,A -85,B 0,C 180,E1 -24648.112,E2 -24648.112} C_VEL
LIN {X 0,Y 136.059,Z 613.7,A -85,B 0,C 180,E1 -24652.581,E2 -24652.581} C_VEL
LIN {X 0,Y 136.282,Z 607.441,A -85,B 0,C 180,E1 -24657.044,E2 -24657.044} C_VEL
LIN {X 0,Y 136.524,Z 600.986,A -85,B 0,C 180,E1 -24660.738,E2 -24660.738} C_VEL
LIN {X 0,Y 136.69,Z 593.041,A -85,B 0,C 180,E1 -24664.423,E2 -24664.423} C_VEL
LIN {X 0,Y 136.98,Z 582.28,A -85,B 0,C 180,E1 -24668.483,E2 -24668.483} C_VEL
LIN {X 0,Y 137.63,Z 571.369,A -85,B 0,C 180,E1 -24671.786,E2 -24671.786} C_VEL
LIN {X 0,Y 138.573,Z 556.125,A -85,B 0,C 180,E1 -24675.553,E2 -24675.553} C_VEL
LIN {X 0,Y 138.591,Z 554.66,A -85,B 0,C 180,E1 -24676.383,E2 -24676.383} C_VEL
LIN {X 0,Y 139.292,Z 554.53,A -85,B 0,C 180,E1 -24677.622,E2 -24677.622} C_VEL
LIN {X 0,Y 141.141,Z 553.024,A -85,B 0,C 180,E1 -24678.89,E2 -24678.89} C_VEL
LIN {X 0,Y 143.747,Z 549.969,A -85,B 0,C 180,E1 -24680.014,E2 -24680.014} C_VEL
LIN {X 0,Y 147.473,Z 547.313,A -85,B 0,C 180,E1 -24682.411,E2 -24682.411} C_VEL
LIN {X 0,Y 150.449,Z 543.948,A -85,B 0,C 180,E1 -24683.642,E2 -24683.642} C_VEL
LIN {X 0,Y 153.037,Z 540.308,A -85,B 0,C 180,E1 -24684.413,E2 -24684.413} C_VEL
LIN {X 0,Y 154.658,Z 538.396,A -85,B 0,C 180,E1 -24685.063,E2 -24685.063} C_VEL
LIN {X 0,Y 156.055,Z 537.181,A -85,B 0,C 180,E1 -24685.742,E2 -24685.742} C_VEL
LIN {X 0,Y 159.133,Z 533.53,A -85,B 0,C 180,E1 -24686.916,E2 -24686.916} C_VEL
LIN {X 0,Y 162.538,Z 528.125,A -85,B 0,C 180,E1 -24687.874,E2 -24687.874} C_VEL
LIN {X 0,Y 166.737,Z 519.066,A -85,B 0,C 180,E1 -24688.79,E2 -24688.79} C_VEL
LIN {X 0,Y 167.235,Z 518.016,A -85,B 0,C 180,E1 -24688.922,E2 -24688.922} C_VEL
LIN {X 0,Y 170.383,Z 513.417,A -85,B 0,C 180,E1 -24690.129,E2 -24690.129} C_VEL
LIN {X 0,Y 173.456,Z 507.256,A -85,B 0,C 180,E1 -24691.139,E2 -24691.139} C_VEL
LIN {X 0,Y 176.707,Z 498.223,A -85,B 0,C 180,E1 -24692.109,E2 -24692.109} C_VEL
LIN {X 0,Y 181.019,Z 483.946,A -85,B 0,C 180,E1 -24693.224,E2 -24693.224} C_VEL
LIN {X 0,Y 184.869,Z 477.239,A -85,B 0,C 180,E1 -24694.558,E2 -24694.558} C_VEL
LIN {X 0,Y 188.023,Z 470.368,A -85,B 0,C 180,E1 -24695.49,E2 -24695.49} C_VEL
LIN {X 0,Y 190.058,Z 465.184,A -85,B 0,C 180,E1 -24696.017,E2 -24696.017} C_VEL
LIN {X 0,Y 191.447,Z 463.138,A -85,B 0,C 180,E1 -24696.459,E2 -24696.459} C_VEL
LIN {X 0,Y 187.614,Z 510.371,A -85,B 0,C 180,E1 -24697.952,E2 -24697.952} C_VEL
LIN {X 0,Y 185.416,Z 524.37,A -85,B 0,C 180,E1 -24698.682,E2 -24698.682} C_VEL
LIN {X 0,Y 182.185,Z 538.261,A -85,B 0,C 180,E1 -24699.722,E2 -24699.722} C_VEL
LIN {X 0,Y 178.395,Z 551.188,A -85,B 0,C 180,E1 -24701.107,E2 -24701.107} C_VEL
LIN {X 0,Y 173.81,Z 563.733,A -85,B 0,C 180,E1 -24702.868,E2 -24702.868} C_VEL
LIN {X 0,Y 168.704,Z 575.683,A -85,B 0,C 180,E1 -24705.089,E2 -24705.089} C_VEL
LIN {X 0,Y 163.841,Z 585.686,A -85,B 0,C 180,E1 -24707.496,E2 -24707.496} C_VEL
LIN {X 0,Y 157.993,Z 596.124,A -85,B 0,C 180,E1 -24710.659,E2 -24710.659} C_VEL
LIN {X 0,Y 152.683,Z 604.735,A -85,B 0,C 180,E1 -24714.06,E2 -24714.06} C_VEL
LIN {X 0,Y 147.227,Z 612.987,A -85,B 0,C 180,E1 -24718.322,E2 -24718.322} C_VEL
LIN {X 0,Y 143.055,Z 618.994,A -85,B 0,C 180,E1 -24722.393,E2 -24722.393} C_VEL
LIN {X 0,Y 139.08,Z 624.879,A -85,B 0,C 180,E1 -24727.725,E2 -24727.725} C_VEL
LIN {X 0,Y 136.571,Z 628.374,A -85,B 0,C 180,E1 -24732.012,E2 -24732.012} C_VEL
LIN {X 0,Y 134.479,Z 631.784,A -85,B 0,C 180,E1 -24737.93,E2 -24737.93} C_VEL
LIN {X 0,Y 133.549,Z 633.809,A -85,B 0,C 180,E1 -24743.955,E2 -24743.955} C_VEL
LIN {X 0,Y 133.419,Z 634.499,A -85,B 0,C 180,E1 -24749.996,E2 -24749.996} C_VEL
LIN {X 0,Y 133.546,Z 633.861,A -85,B 0,C 180,E1 -24756.038,E2 -24756.038} C_VEL
LIN {X 0,Y 134.472,Z 631.883,A -85,B 0,C 180,E1 -24762.063,E2 -24762.063} C_VEL
LIN {X 0,Y 136.548,Z 628.516,A -85,B 0,C 180,E1 -24767.984,E2 -24767.984} C_VEL
LIN {X 0,Y 140,Z 623.66,A -85,B 0,C 180,E1 -24773.674,E2 -24773.674} C_VEL
LIN {X 0,Y 143.615,Z 618.348,A -85,B 0,C 180,E1 -24778.253,E2 -24778.253} C_VEL
LIN {X 0,Y 148.625,Z 611.063,A -85,B 0,C 180,E1 -24782.938,E2 -24782.938} C_VEL
LIN {X 0,Y 154.307,Z 602.377,A -85,B 0,C 180,E1 -24787.115,E2 -24787.115} C_VEL
LIN {X 0,Y 159.784,Z 593.29,A -85,B 0,C 180,E1 -24790.444,E2 -24790.444} C_VEL
LIN {X 0,Y 165.408,Z 582.962,A -85,B 0,C 180,E1 -24793.369,E2 -24793.369} C_VEL
LIN {X 0,Y 170.429,Z 572.26,A -85,B 0,C 180,E1 -24795.761,E2 -24795.761} C_VEL
LIN {X 0,Y 175.397,Z 560.184,A -85,B 0,C 180,E1 -24797.835,E2 -24797.835} C_VEL
LIN {X 0,Y 179.425,Z 548.556,A -85,B 0,C 180,E1 -24799.363,E2 -24799.363} C_VEL
LIN {X 0,Y 183.231,Z 534.805,A -85,B 0,C 180,E1 -24800.738,E2 -24800.738} C_VEL
LIN {X 0,Y 186.289,Z 520.211,A -85,B 0,C 180,E1 -24801.732,E2 -24801.732} C_VEL
LIN {X 0,Y 188.272,Z 506.15,A -85,B 0,C 180,E1 -24802.339,E2 -24802.339} C_VEL
LIN {X 0,Y 191.896,Z 459.625,A -85,B 0,C 180,E1 -24803.792,E2 -24803.792} C_VEL
LIN {X 0,Y 187.412,Z 448.407,A -85,B 0,C 180,E1 -24806.462,E2 -24806.462} C_VEL
LIN {X 0,Y 184.191,Z 441.618,A -85,B 0,C 180,E1 -24808.496,E2 -24808.496} C_VEL
